KUKA KRL program: EPS_2_251349_MH86A_A_20250929014656.src

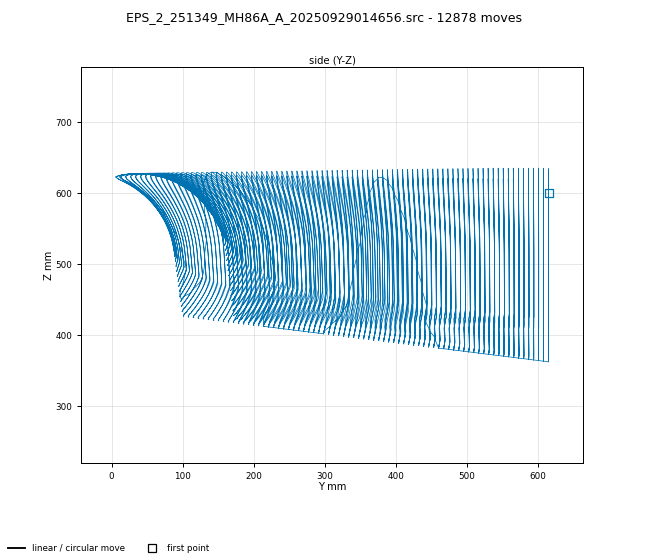
[picture p0: tool path of EPS_2_251349_MH86A_A_20250929014656.src, 12878 of 12880 moves have a stored position in this frame; points joined in program order, loops and branches not executed]
&ACCESS RVP
&REL 4
&COMMENT QRS 19112012
&PARAM EDITMASK = *
DEF PART()
EXT BAS (BAS_COMMAND :IN,REAL :IN )
INT I
BAS (#INITMOV,0 )

;KUKA QRS Post kuka4.cps  Date:22-06-2017 !

File_ID=2862

QRS_PRE_INIT()

;Init var - Until changes are made in qrs_pre_init
Outlet_Square_prg=0
Inlet_1_Square_prg=0
Inlet_2_Square_prg=0
Inlet_3_Square_prg=0
Inlet_4_Square_prg=0
Inlet_5_Square_prg=0

Outlet_1={X 0.000, Y 530.070, Z 534.500, B 0.000, E1 0.000 }
Inlet_1={X 0.000, Y 531.140, Z 519.500, B 0.000, E1 193.000 }
Outlet_1_type=201
Inlet_1_type=201
;QRS#1=Sidecore dimensions
;QRS#2=200-8" PVC SDR 35
;QRS#3=200-8" PVC SDR 35
;QRS#4=
;QRS#5=
;QRS#6=
;QRS#7=
;QRS#8=
;QRS#9=12-08 PSX
;QRS#10=12-08 PSX
;QRS#11=
;QRS#12=
;QRS#13=
;QRS#14=
;QRS#15=
;QRS#16=1220x127x914 3'
;QRS#17=EPS Height
;QRS#18=635
;QRS#19=*
;QRS#20= UPDATED VERSION 22-06-2017
;QRS#21=*
Outlet_Square=0100
Inlet_1_Square=0100
Inlet_2_Square=0
Inlet_3_Square=0
Inlet_4_Square=0
Inlet_5_Square=0
Mill_Square=1
Outlet_Square_Prg=204
Inlet_1_Square_prg=204

QRS_INIT()

$ADVANCE=5

; T1
PTP {E1 173.597,E2 173.597}
PTP {X 0,Y 615.506,A -85,B 0,C 180,E1 173.597,E2 173.597,E3 0,E4 0,E5 0,E6 0}
QRS_SPEED_INIT()
LIN {X 0,Y 615.506,Z 600,A -85,B 0,C 180,E1 173.597,E2 173.597,E3 0,E4 0,E5 0,E6 0} C_VEL
LIN {X 0,Y 615.506,Z 372.373,A -85,B 0,C 180,E1 173.597,E2 173.597} C_VEL
LIN {X 0,Y 615.506,Z 364.191,A -85,B 0,C 180,E1 173.597,E2 173.597} C_VEL
LIN {X 0,Y 615.49,Z 362.191,A -85,B 0,C 180,E1 173.411,E2 173.411} C_VEL
LIN {X 0,Y 615.479,Z 362.185,A -85,B 0,C 180,E1 170.801,E2 170.801} C_VEL
LIN {X 0,Y 615.477,Z 362.195,A -85,B 0,C 180,E1 168.139,E2 168.139} C_VEL
LIN {X 0,Y 615.49,Z 362.189,A -85,B 0,C 180,E1 165.451,E2 165.451} C_VEL
LIN {X 0,Y 615.49,Z 362.183,A -85,B 0,C 180,E1 162.73,E2 162.73} C_VEL
LIN {X 0,Y 615.493,Z 362.201,A -85,B 0,C 180,E1 159.967,E2 159.967} C_VEL
LIN {X 0,Y 615.477,Z 362.185,A -85,B 0,C 180,E1 157.155,E2 157.155} C_VEL
LIN {X 0,Y 615.493,Z 362.19,A -85,B 0,C 180,E1 154.428,E2 154.428} C_VEL
LIN {X 0,Y 615.491,Z 362.185,A -85,B 0,C 180,E1 151.547,E2 151.547} C_VEL
LIN {X 0,Y 615.483,Z 362.185,A -85,B 0,C 180,E1 148.913,E2 148.913} C_VEL
LIN {X 0,Y 615.495,Z 362.193,A -85,B 0,C 180,E1 146.463,E2 146.463} C_VEL
LIN {X 0,Y 615.488,Z 362.184,A -85,B 0,C 180,E1 143.575,E2 143.575} C_VEL
LIN {X 0,Y 615.48,Z 362.187,A -85,B 0,C 180,E1 140.938,E2 140.938} C_VEL
LIN {X 0,Y 615.494,Z 362.195,A -85,B 0,C 180,E1 138.527,E2 138.527} C_VEL
LIN {X 0,Y 615.495,Z 362.185,A -85,B 0,C 180,E1 135.851,E2 135.851} C_VEL
LIN {X 0,Y 615.481,Z 362.188,A -85,B 0,C 180,E1 133.047,E2 133.047} C_VEL
LIN {X 0,Y 615.494,Z 362.198,A -85,B 0,C 180,E1 130.605,E2 130.605} C_VEL
LIN {X 0,Y 615.489,Z 362.187,A -85,B 0,C 180,E1 128.012,E2 128.012} C_VEL
LIN {X 0,Y 615.486,Z 362.183,A -85,B 0,C 180,E1 125.615,E2 125.615} C_VEL
LIN {X 0,Y 615.478,Z 362.188,A -85,B 0,C 180,E1 123.236,E2 123.236} C_VEL
LIN {X 0,Y 615.492,Z 362.193,A -85,B 0,C 180,E1 120.919,E2 120.919} C_VEL
LIN {X 0,Y 615.483,Z 362.194,A -85,B 0,C 180,E1 118.449,E2 118.449} C_VEL
LIN {X 0,Y 615.481,Z 362.185,A -85,B 0,C 180,E1 115.567,E2 115.567} C_VEL
LIN {X 0,Y 615.489,Z 362.202,A -85,B 0,C 180,E1 112.844,E2 112.844} C_VEL
LIN {X 0,Y 615.485,Z 362.184,A -85,B 0,C 180,E1 110.033,E2 110.033} C_VEL
LIN {X 0,Y 615.479,Z 362.193,A -85,B 0,C 180,E1 107.271,E2 107.271} C_VEL
LIN {X 0,Y 615.479,Z 362.191,A -85,B 0,C 180,E1 104.549,E2 104.549} C_VEL
LIN {X 0,Y 615.489,Z 362.183,A -85,B 0,C 180,E1 101.861,E2 101.861} C_VEL
LIN {X 0,Y 615.49,Z 362.198,A -85,B 0,C 180,E1 99.199,E2 99.199} C_VEL
LIN {X 0,Y 615.499,Z 362.314,A -85,B 0,C 180,E1 97.058,E2 97.058} C_VEL
LIN {X 0,Y 615.484,Z 376.753,A -85,B 0,C 180,E1 94.749,E2 94.749} C_VEL
LIN {X 0,Y 615.497,Z 394.683,A -85,B 0,C 180,E1 91.963,E2 91.963} C_VEL
LIN {X 0,Y 615.488,Z 408.592,A -85,B 0,C 180,E1 89.857,E2 89.857} C_VEL
LIN {X 0,Y 615.485,Z 410.307,A -85,B 0,C 180,E1 89.796,E2 89.796} C_VEL
LIN {X 0,Y 615.497,Z 515.58,A -85,B 0,C 180,E1 88.548,E2 88.548} C_VEL
LIN {X 0,Y 615.498,Z 527.992,A -85,B 0,C 180,E1 88.283,E2 88.283} C_VEL
LIN {X 0,Y 615.498,Z 540.764,A -85,B 0,C 180,E1 87.873,E2 87.873} C_VEL
LIN {X 0,Y 615.486,Z 552.111,A -85,B 0,C 180,E1 87.382,E2 87.382} C_VEL
LIN {X 0,Y 615.484,Z 563.831,A -85,B 0,C 180,E1 86.727,E2 86.727} C_VEL
LIN {X 0,Y 615.498,Z 574.262,A -85,B 0,C 180,E1 85.99,E2 85.99} C_VEL
LIN {X 0,Y 615.497,Z 584.574,A -85,B 0,C 180,E1 85.088,E2 85.088} C_VEL
LIN {X 0,Y 615.499,Z 593.527,A -85,B 0,C 180,E1 84.102,E2 84.102} C_VEL
LIN {X 0,Y 615.497,Z 600.873,A -85,B 0,C 180,E1 83.1,E2 83.1} C_VEL
LIN {X 0,Y 615.497,Z 606.596,A -85,B 0,C 180,E1 82.125,E2 82.125} C_VEL
LIN {X 0,Y 615.497,Z 611.188,A -85,B 0,C 180,E1 81.133,E2 81.133} C_VEL
LIN {X 0,Y 615.498,Z 614.685,A -85,B 0,C 180,E1 80.138,E2 80.138} C_VEL
LIN {X 0,Y 615.494,Z 617.25,A -85,B 0,C 180,E1 79.109,E2 79.109} C_VEL
LIN {X 0,Y 615.496,Z 618.726,A -85,B 0,C 180,E1 78.14,E2 78.14} C_VEL
LIN {X 0,Y 615.497,Z 619.266,A -85,B 0,C 180,E1 77.47,E2 77.47} C_VEL
LIN {X 0,Y 615.496,Z 619.357,A -85,B 0,C 180,E1 76.799,E2 76.799} C_VEL
LIN {X 0,Y 615.496,Z 619.007,A -85,B 0,C 180,E1 76.065,E2 76.065} C_VEL
LIN {X 0,Y 615.495,Z 618.351,A -85,B 0,C 180,E1 75.452,E2 75.452} C_VEL
LIN {X 0,Y 615.495,Z 617.194,A -85,B 0,C 180,E1 74.775,E2 74.775} C_VEL
LIN {X 0,Y 615.493,Z 614.033,A -85,B 0,C 180,E1 73.568,E2 73.568} C_VEL
LIN {X 0,Y 615.499,Z 609.514,A -85,B 0,C 180,E1 72.387,E2 72.387} C_VEL
LIN {X 0,Y 615.496,Z 604.234,A -85,B 0,C 180,E1 71.355,E2 71.355} C_VEL
LIN {X 0,Y 615.496,Z 597.453,A -85,B 0,C 180,E1 70.316,E2 70.316} C_VEL
LIN {X 0,Y 615.494,Z 588.884,A -85,B 0,C 180,E1 69.27,E2 69.27} C_VEL
LIN {X 0,Y 615.497,Z 579.965,A -85,B 0,C 180,E1 68.393,E2 68.393} C_VEL
LIN {X 0,Y 615.495,Z 568.994,A -85,B 0,C 180,E1 67.528,E2 67.528} C_VEL
LIN {X 0,Y 615.484,Z 558.946,A -85,B 0,C 180,E1 66.89,E2 66.89} C_VEL
LIN {X 0,Y 615.5,Z 546.63,A -85,B 0,C 180,E1 66.274,E2 66.274} C_VEL
LIN {X 0,Y 615.497,Z 533.761,A -85,B 0,C 180,E1 65.794,E2 65.794} C_VEL
LIN {X 0,Y 615.495,Z 520.923,A -85,B 0,C 180,E1 65.46,E2 65.46} C_VEL
LIN {X 0,Y 615.497,Z 505.869,A -85,B 0,C 180,E1 65.235,E2 65.235} C_VEL
LIN {X 0,Y 615.487,Z 409.668,A -85,B 0,C 180,E1 64.103,E2 64.103} C_VEL
LIN {X 0,Y 615.488,Z 408.193,A -85,B 0,C 180,E1 64.012,E2 64.012} C_VEL
LIN {X 0,Y 615.498,Z 389.57,A -85,B 0,C 180,E1 61.157,E2 61.157} C_VEL
LIN {X 0,Y 615.488,Z 371.358,A -85,B 0,C 180,E1 58.316,E2 58.316} C_VEL
LIN {X 0,Y 615.493,Z 362.338,A -85,B 0,C 180,E1 56.863,E2 56.863} C_VEL
LIN {X 0,Y 615.489,Z 362.184,A -85,B 0,C 180,E1 54.166,E2 54.166} C_VEL
LIN {X 0,Y 615.482,Z 362.184,A -85,B 0,C 180,E1 51.932,E2 51.932} C_VEL
LIN {X 0,Y 615.483,Z 362.187,A -85,B 0,C 180,E1 49.394,E2 49.394} C_VEL
LIN {X 0,Y 615.495,Z 362.197,A -85,B 0,C 180,E1 46.757,E2 46.757} C_VEL
LIN {X 0,Y 615.482,Z 362.184,A -85,B 0,C 180,E1 43.998,E2 43.998} C_VEL
LIN {X 0,Y 615.485,Z 362.186,A -85,B 0,C 180,E1 41.474,E2 41.474} C_VEL
LIN {X 0,Y 615.497,Z 362.2,A -85,B 0,C 180,E1 38.904,E2 38.904} C_VEL
LIN {X 0,Y 615.493,Z 362.186,A -85,B 0,C 180,E1 36.424,E2 36.424} C_VEL
LIN {X 0,Y 615.484,Z 362.186,A -85,B 0,C 180,E1 33.536,E2 33.536} C_VEL
LIN {X 0,Y 615.493,Z 362.2,A -85,B 0,C 180,E1 30.919,E2 30.919} C_VEL
LIN {X 0,Y 615.495,Z 362.185,A -85,B 0,C 180,E1 28.454,E2 28.454} C_VEL
LIN {X 0,Y 615.479,Z 362.186,A -85,B 0,C 180,E1 25.716,E2 25.716} C_VEL
LIN {X 0,Y 615.489,Z 362.196,A -85,B 0,C 180,E1 22.844,E2 22.844} C_VEL
LIN {X 0,Y 615.479,Z 362.184,A -85,B 0,C 180,E1 20.033,E2 20.033} C_VEL
LIN {X 0,Y 615.496,Z 362.193,A -85,B 0,C 180,E1 17.27,E2 17.27} C_VEL
LIN {X 0,Y 615.493,Z 362.186,A -85,B 0,C 180,E1 14.549,E2 14.549} C_VEL
LIN {X 0,Y 615.476,Z 362.186,A -85,B 0,C 180,E1 11.861,E2 11.861} C_VEL
LIN {X 0,Y 615.496,Z 362.198,A -85,B 0,C 180,E1 9.199,E2 9.199} C_VEL
LIN {X 0,Y 615.495,Z 362.184,A -85,B 0,C 180,E1 6.557,E2 6.557} C_VEL
LIN {X 0,Y 615.476,Z 362.186,A -85,B 0,C 180,E1 3.929,E2 3.929} C_VEL
LIN {X 0,Y 615.496,Z 362.195,A -85,B 0,C 180,E1 1.309,E2 1.309} C_VEL
LIN {X 0,Y 615.491,Z 362.187,A -85,B 0,C 180,E1 -1.309,E2 -1.309} C_VEL
LIN {X 0,Y 615.476,Z 362.185,A -85,B 0,C 180,E1 -3.929,E2 -3.929} C_VEL
LIN {X 0,Y 615.497,Z 362.194,A -85,B 0,C 180,E1 -6.598,E2 -6.598} C_VEL
LIN {X 0,Y 615.486,Z 362.189,A -85,B 0,C 180,E1 -9.199,E2 -9.199} C_VEL
LIN {X 0,Y 615.478,Z 362.185,A -85,B 0,C 180,E1 -11.861,E2 -11.861} C_VEL
LIN {X 0,Y 615.497,Z 362.194,A -85,B 0,C 180,E1 -14.549,E2 -14.549} C_VEL
LIN {X 0,Y 615.493,Z 362.185,A -85,B 0,C 180,E1 -17.27,E2 -17.27} C_VEL
LIN {X 0,Y 615.479,Z 362.186,A -85,B 0,C 180,E1 -20.033,E2 -20.033} C_VEL
LIN {X 0,Y 615.492,Z 362.196,A -85,B 0,C 180,E1 -22.844,E2 -22.844} C_VEL
LIN {X 0,Y 615.477,Z 362.184,A -85,B 0,C 180,E1 -25.716,E2 -25.716} C_VEL
LIN {X 0,Y 615.497,Z 362.194,A -85,B 0,C 180,E1 -28.454,E2 -28.454} C_VEL
LIN {X 0,Y 615.49,Z 362.188,A -85,B 0,C 180,E1 -31.089,E2 -31.089} C_VEL
LIN {X 0,Y 615.484,Z 362.183,A -85,B 0,C 180,E1 -33.536,E2 -33.536} C_VEL
LIN {X 0,Y 615.495,Z 362.195,A -85,B 0,C 180,E1 -36.424,E2 -36.424} C_VEL
LIN {X 0,Y 615.488,Z 362.188,A -85,B 0,C 180,E1 -39.064,E2 -39.064} C_VEL
LIN {X 0,Y 615.485,Z 362.183,A -85,B 0,C 180,E1 -41.474,E2 -41.474} C_VEL
LIN {X 0,Y 615.491,Z 362.189,A -85,B 0,C 180,E1 -44.149,E2 -44.149} C_VEL
LIN {X 0,Y 615.489,Z 362.189,A -85,B 0,C 180,E1 -46.953,E2 -46.953} C_VEL
LIN {X 0,Y 615.482,Z 362.183,A -85,B 0,C 180,E1 -49.394,E2 -49.394} C_VEL
LIN {X 0,Y 615.484,Z 362.188,A -85,B 0,C 180,E1 -51.989,E2 -51.989} C_VEL
LIN {X 0,Y 615.496,Z 362.198,A -85,B 0,C 180,E1 -54.386,E2 -54.386} C_VEL
LIN {X 0,Y 615.488,Z 362.192,A -85,B 0,C 180,E1 -56.765,E2 -56.765} C_VEL
LIN {X 0,Y 615.495,Z 362.183,A -85,B 0,C 180,E1 -59.082,E2 -59.082} C_VEL
LIN {X 0,Y 615.477,Z 362.185,A -85,B 0,C 180,E1 -61.552,E2 -61.552} C_VEL
LIN {X 0,Y 615.498,Z 362.2,A -85,B 0,C 180,E1 -64.43,E2 -64.43} C_VEL
LIN {X 0,Y 615.488,Z 362.183,A -85,B 0,C 180,E1 -67.156,E2 -67.156} C_VEL
LIN {X 0,Y 615.495,Z 362.441,A -85,B 0,C 180,E1 -68.481,E2 -68.481} C_VEL
LIN {X 0,Y 615.495,Z 380.964,A -85,B 0,C 180,E1 -71.182,E2 -71.182} C_VEL
LIN {X 0,Y 615.489,Z 401.427,A -85,B 0,C 180,E1 -74.095,E2 -74.095} C_VEL
LIN {X 0,Y 615.497,Z 422.521,A -85,B 0,C 180,E1 -77.051,E2 -77.051} C_VEL
LIN {X 0,Y 615.497,Z 423.747,A -85,B 0,C 180,E1 -77.135,E2 -77.135} C_VEL
LIN {X 0,Y 615.498,Z 530.85,A -85,B 0,C 180,E1 -78.411,E2 -78.411} C_VEL
LIN {X 0,Y 615.498,Z 543.356,A -85,B 0,C 180,E1 -78.682,E2 -78.682} C_VEL
LIN {X 0,Y 615.496,Z 556.503,A -85,B 0,C 180,E1 -79.109,E2 -79.109} C_VEL
LIN {X 0,Y 615.483,Z 568.485,A -85,B 0,C 180,E1 -79.64,E2 -79.64} C_VEL
LIN {X 0,Y 615.487,Z 580.001,A -85,B 0,C 180,E1 -80.304,E2 -80.304} C_VEL
LIN {X 0,Y 615.499,Z 590.345,A -85,B 0,C 180,E1 -81.05,E2 -81.05} C_VEL
LIN {X 0,Y 615.497,Z 598.815,A -85,B 0,C 180,E1 -81.794,E2 -81.794} C_VEL
LIN {X 0,Y 615.498,Z 606.609,A -85,B 0,C 180,E1 -82.62,E2 -82.62} C_VEL
LIN {X 0,Y 615.496,Z 614.205,A -85,B 0,C 180,E1 -83.608,E2 -83.608} C_VEL
LIN {X 0,Y 615.499,Z 621.206,A -85,B 0,C 180,E1 -84.759,E2 -84.759} C_VEL
LIN {X 0,Y 615.493,Z 625.853,A -85,B 0,C 180,E1 -85.744,E2 -85.744} C_VEL
LIN {X 0,Y 615.495,Z 629.399,A -85,B 0,C 180,E1 -86.727,E2 -86.727} C_VEL
LIN {X 0,Y 615.497,Z 631.233,A -85,B 0,C 180,E1 -87.382,E2 -87.382} C_VEL
LIN {X 0,Y 615.497,Z 632.608,A -85,B 0,C 180,E1 -88.037,E2 -88.037} C_VEL
LIN {X 0,Y 615.496,Z 634.174,A -85,B 0,C 180,E1 -89.346,E2 -89.346} C_VEL
LIN {X 0,Y 615.494,Z 634.389,A -85,B 0,C 180,E1 -90,E2 -90} C_VEL
LIN {X 0,Y 615.496,Z 633.58,A -85,B 0,C 180,E1 -91.309,E2 -91.309} C_VEL
LIN {X 0,Y 615.497,Z 632.608,A -85,B 0,C 180,E1 -91.963,E2 -91.963} C_VEL
LIN {X 0,Y 615.497,Z 631.233,A -85,B 0,C 180,E1 -92.618,E2 -92.618} C_VEL
LIN {X 0,Y 615.496,Z 628.349,A -85,B 0,C 180,E1 -93.601,E2 -93.601} C_VEL
LIN {X 0,Y 615.498,Z 624.441,A -85,B 0,C 180,E1 -94.585,E2 -94.585} C_VEL
LIN {X 0,Y 615.499,Z 619.405,A -85,B 0,C 180,E1 -95.57,E2 -95.57} C_VEL
LIN {X 0,Y 615.497,Z 612.87,A -85,B 0,C 180,E1 -96.583,E2 -96.583} C_VEL
LIN {X 0,Y 615.497,Z 605.133,A -85,B 0,C 180,E1 -97.545,E2 -97.545} C_VEL
LIN {X 0,Y 615.498,Z 597.045,A -85,B 0,C 180,E1 -98.371,E2 -98.371} C_VEL
LIN {X 0,Y 615.499,Z 587.168,A -85,B 0,C 180,E1 -99.199,E2 -99.199} C_VEL
LIN {X 0,Y 615.487,Z 575.982,A -85,B 0,C 180,E1 -99.945,E2 -99.945} C_VEL
LIN {X 0,Y 615.486,Z 565.024,A -85,B 0,C 180,E1 -100.527,E2 -100.527} C_VEL
LIN {X 0,Y 615.499,Z 552.418,A -85,B 0,C 180,E1 -101.042,E2 -101.042} C_VEL
LIN {X 0,Y 615.499,Z 540.066,A -85,B 0,C 180,E1 -101.401,E2 -101.401} C_VEL
LIN {X 0,Y 615.499,Z 526.468,A -85,B 0,C 180,E1 -101.652,E2 -101.652} C_VEL
LIN {X 0,Y 615.496,Z 423.736,A -85,B 0,C 180,E1 -102.865,E2 -102.865} C_VEL
LIN {X 0,Y 615.497,Z 422.518,A -85,B 0,C 180,E1 -102.949,E2 -102.949} C_VEL
LIN {X 0,Y 615.489,Z 401.425,A -85,B 0,C 180,E1 -105.905,E2 -105.905} C_VEL
LIN {X 0,Y 615.495,Z 380.962,A -85,B 0,C 180,E1 -108.818,E2 -108.818} C_VEL
LIN {X 0,Y 615.496,Z 362.439,A -85,B 0,C 180,E1 -111.519,E2 -111.519} C_VEL
LIN {X 0,Y 615.488,Z 362.184,A -85,B 0,C 180,E1 -112.844,E2 -112.844} C_VEL
LIN {X 0,Y 615.498,Z 362.194,A -85,B 0,C 180,E1 -115.715,E2 -115.715} C_VEL
LIN {X 0,Y 615.477,Z 362.185,A -85,B 0,C 180,E1 -118.448,E2 -118.448} C_VEL
LIN {X 0,Y 615.492,Z 362.19,A -85,B 0,C 180,E1 -121.086,E2 -121.086} C_VEL
LIN {X 0,Y 615.484,Z 362.186,A -85,B 0,C 180,E1 -124.022,E2 -124.022} C_VEL
LIN {X 0,Y 615.479,Z 362.185,A -85,B 0,C 180,E1 -126.425,E2 -126.425} C_VEL
LIN {X 0,Y 615.493,Z 362.193,A -85,B 0,C 180,E1 -129.062,E2 -129.062} C_VEL
LIN {X 0,Y 615.494,Z 362.194,A -85,B 0,C 180,E1 -131.472,E2 -131.472} C_VEL
LIN {X 0,Y 615.478,Z 362.185,A -85,B 0,C 180,E1 -134.149,E2 -134.149} C_VEL
LIN {X 0,Y 615.494,Z 362.194,A -85,B 0,C 180,E1 -136.951,E2 -136.951} C_VEL
LIN {X 0,Y 615.486,Z 362.184,A -85,B 0,C 180,E1 -139.91,E2 -139.91} C_VEL
LIN {X 0,Y 615.494,Z 362.191,A -85,B 0,C 180,E1 -142.758,E2 -142.758} C_VEL
LIN {X 0,Y 615.49,Z 362.192,A -85,B 0,C 180,E1 -145.298,E2 -145.298} C_VEL
LIN {X 0,Y 615.493,Z 362.183,A -85,B 0,C 180,E1 -147.667,E2 -147.667} C_VEL
LIN {X 0,Y 615.489,Z 362.192,A -85,B 0,C 180,E1 -150.594,E2 -150.594} C_VEL
LIN {X 0,Y 615.493,Z 362.183,A -85,B 0,C 180,E1 -153.556,E2 -153.556} C_VEL
LIN {X 0,Y 615.485,Z 362.191,A -85,B 0,C 180,E1 -156.443,E2 -156.443} C_VEL
LIN {X 0,Y 615.479,Z 362.189,A -85,B 0,C 180,E1 -159.269,E2 -159.269} C_VEL
LIN {X 0,Y 615.477,Z 362.187,A -85,B 0,C 180,E1 -162.043,E2 -162.043} C_VEL
LIN {X 0,Y 615.486,Z 362.199,A -85,B 0,C 180,E1 -164.774,E2 -164.774} C_VEL
LIN {X 0,Y 615.484,Z 362.184,A -85,B 0,C 180,E1 -167.47,E2 -167.47} C_VEL
LIN {X 0,Y 615.477,Z 362.192,A -85,B 0,C 180,E1 -170.138,E2 -170.138} C_VEL
LIN {X 0,Y 615.483,Z 362.194,A -85,B 0,C 180,E1 -172.784,E2 -172.784} C_VEL
LIN {X 0,Y 615.491,Z 362.182,A -85,B 0,C 180,E1 -175.415,E2 -175.415} C_VEL
LIN {X 0,Y 615.478,Z 362.193,A -85,B 0,C 180,E1 -178.037,E2 -178.037} C_VEL
LIN {X 0,Y 615.484,Z 362.194,A -85,B 0,C 180,E1 -180.654,E2 -180.654} C_VEL
LIN {X 0,Y 615.485,Z 362.183,A -85,B 0,C 180,E1 -183.273,E2 -183.273} C_VEL
LIN {X 0,Y 615.481,Z 362.192,A -85,B 0,C 180,E1 -185.899,E2 -185.899} C_VEL
LIN {X 0,Y 615.49,Z 362.191,A -85,B 0,C 180,E1 -186.589,E2 -186.589} C_VEL
LIN {X 0,Y 614.809,Z 362.332,A -85,B 0,C 180,E1 -187.135,E2 -187.135} C_VEL
LIN {X 0,Y 611.969,Z 362.756,A -85,B 0,C 180,E1 -188.021,E2 -188.021} C_VEL
LIN {X 0,Y 609.575,Z 363.062,A -85,B 0,C 180,E1 -188.733,E2 -188.733} C_VEL
LIN {X 0,Y 608.54,Z 363.178,A -85,B 0,C 180,E1 -189.283,E2 -189.283} C_VEL
LIN {X 0,Y 608.452,Z 363.188,A -85,B 0,C 180,E1 -189.469,E2 -189.469} C_VEL
LIN {X 0,Y 608.455,Z 363.195,A -85,B 0,C 180,E1 -192,E2 -192} C_VEL
LIN {X 0,Y 608.476,Z 363.186,A -85,B 0,C 180,E1 -194.72,E2 -194.72} C_VEL
LIN {X 0,Y 608.456,Z 363.189,A -85,B 0,C 180,E1 -197.476,E2 -197.476} C_VEL
LIN {X 0,Y 608.466,Z 363.192,A -85,B 0,C 180,E1 -200.274,E2 -200.274} C_VEL
LIN {X 0,Y 608.457,Z 363.19,A -85,B 0,C 180,E1 -202.478,E2 -202.478} C_VEL
LIN {X 0,Y 608.453,Z 363.189,A -85,B 0,C 180,E1 -204.571,E2 -204.571} C_VEL
LIN {X 0,Y 608.474,Z 363.186,A -85,B 0,C 180,E1 -207.208,E2 -207.208} C_VEL
LIN {X 0,Y 608.475,Z 363.193,A -85,B 0,C 180,E1 -209.974,E2 -209.974} C_VEL
LIN {X 0,Y 608.463,Z 363.187,A -85,B 0,C 180,E1 -212.524,E2 -212.524} C_VEL
LIN {X 0,Y 608.443,Z 363.192,A -85,B 0,C 180,E1 -215.278,E2 -215.278} C_VEL
LIN {X 0,Y 608.473,Z 363.195,A -85,B 0,C 180,E1 -217.746,E2 -217.746} C_VEL
LIN {X 0,Y 608.451,Z 363.189,A -85,B 0,C 180,E1 -220.33,E2 -220.33} C_VEL
LIN {X 0,Y 608.453,Z 363.189,A -85,B 0,C 180,E1 -222.96,E2 -222.96} C_VEL
LIN {X 0,Y 608.458,Z 363.194,A -85,B 0,C 180,E1 -225.736,E2 -225.736} C_VEL
LIN {X 0,Y 608.457,Z 363.187,A -85,B 0,C 180,E1 -228.658,E2 -228.658} C_VEL
LIN {X 0,Y 608.47,Z 363.195,A -85,B 0,C 180,E1 -231.413,E2 -231.413} C_VEL
LIN {X 0,Y 608.478,Z 363.187,A -85,B 0,C 180,E1 -233.951,E2 -233.951} C_VEL
LIN {X 0,Y 608.464,Z 363.186,A -85,B 0,C 180,E1 -236.33,E2 -236.33} C_VEL
LIN {X 0,Y 608.46,Z 363.188,A -85,B 0,C 180,E1 -238.731,E2 -238.731} C_VEL
LIN {X 0,Y 608.475,Z 363.194,A -85,B 0,C 180,E1 -241.38,E2 -241.38} C_VEL
LIN {X 0,Y 608.471,Z 363.185,A -85,B 0,C 180,E1 -244.279,E2 -244.279} C_VEL
LIN {X 0,Y 608.45,Z 363.193,A -85,B 0,C 180,E1 -246.876,E2 -246.876} C_VEL
LIN {X 0,Y 608.46,Z 363.188,A -85,B 0,C 180,E1 -249.726,E2 -249.726} C_VEL
LIN {X 0,Y 608.451,Z 363.19,A -85,B 0,C 180,E1 -252.524,E2 -252.524} C_VEL
LIN {X 0,Y 608.47,Z 363.191,A -85,B 0,C 180,E1 -255.28,E2 -255.28} C_VEL
LIN {X 0,Y 608.462,Z 363.186,A -85,B 0,C 180,E1 -258,E2 -258} C_VEL
LIN {X 0,Y 608.474,Z 363.191,A -85,B 0,C 180,E1 -260.694,E2 -260.694} C_VEL
LIN {X 0,Y 608.486,Z 363.376,A -85,B 0,C 180,E1 -262.889,E2 -262.889} C_VEL
LIN {X 0,Y 608.498,Z 377.808,A -85,B 0,C 180,E1 -265.197,E2 -265.197} C_VEL
LIN {X 0,Y 608.499,Z 395.794,A -85,B 0,C 180,E1 -268.014,E2 -268.014} C_VEL
LIN {X 0,Y 608.48,Z 408.761,A -85,B 0,C 180,E1 -270,E2 -270} C_VEL
LIN {X 0,Y 608.563,Z 410.777,A -85,B 0,C 180,E1 -270.062,E2 -270.062} C_VEL
LIN {X 0,Y 608.557,Z 516.027,A -85,B 0,C 180,E1 -271.323,E2 -271.323} C_VEL
LIN {X 0,Y 608.56,Z 529.053,A -85,B 0,C 180,E1 -271.613,E2 -271.613} C_VEL
LIN {X 0,Y 608.519,Z 541.614,A -85,B 0,C 180,E1 -272.027,E2 -272.027} C_VEL
LIN {X 0,Y 608.512,Z 553.646,A -85,B 0,C 180,E1 -272.565,E2 -272.565} C_VEL
LIN {X 0,Y 608.483,Z 565.068,A -85,B 0,C 180,E1 -273.228,E2 -273.228} C_VEL
LIN {X 0,Y 608.472,Z 575.378,A -85,B 0,C 180,E1 -273.974,E2 -273.974} C_VEL
LIN {X 0,Y 608.464,Z 584.735,A -85,B 0,C 180,E1 -274.803,E2 -274.803} C_VEL
LIN {X 0,Y 608.459,Z 593.778,A -85,B 0,C 180,E1 -275.8,E2 -275.8} C_VEL
LIN {X 0,Y 608.461,Z 601.1,A -85,B 0,C 180,E1 -276.799,E2 -276.799} C_VEL
LIN {X 0,Y 608.45,Z 606.08,A -85,B 0,C 180,E1 -277.633,E2 -277.633} C_VEL
LIN {X 0,Y 608.427,Z 610.93,A -85,B 0,C 180,E1 -278.636,E2 -278.636} C_VEL
LIN {X 0,Y 608.429,Z 614.661,A -85,B 0,C 180,E1 -279.642,E2 -279.642} C_VEL
LIN {X 0,Y 608.45,Z 618.005,A -85,B 0,C 180,E1 -280.946,E2 -280.946} C_VEL
LIN {X 0,Y 608.44,Z 619.506,A -85,B 0,C 180,E1 -282,E2 -282} C_VEL
LIN {X 0,Y 608.418,Z 619.92,A -85,B 0,C 180,E1 -282.678,E2 -282.678} C_VEL
LIN {X 0,Y 608.442,Z 619.573,A -85,B 0,C 180,E1 -284.006,E2 -284.006} C_VEL
LIN {X 0,Y 608.418,Z 618.715,A -85,B 0,C 180,E1 -284.721,E2 -284.721} C_VEL
LIN {X 0,Y 608.419,Z 617.443,A -85,B 0,C 180,E1 -285.407,E2 -285.407} C_VEL
LIN {X 0,Y 608.424,Z 614.45,A -85,B 0,C 180,E1 -286.515,E2 -286.515} C_VEL
LIN {X 0,Y 608.429,Z 610.832,A -85,B 0,C 180,E1 -287.477,E2 -287.477} C_VEL
LIN {X 0,Y 608.443,Z 606.182,A -85,B 0,C 180,E1 -288.438,E2 -288.438} C_VEL
LIN {X 0,Y 608.451,Z 599.223,A -85,B 0,C 180,E1 -289.57,E2 -289.57} C_VEL
LIN {X 0,Y 608.459,Z 591.706,A -85,B 0,C 180,E1 -290.54,E2 -290.54} C_VEL
LIN {X 0,Y 608.467,Z 582.342,A -85,B 0,C 180,E1 -291.513,E2 -291.513} C_VEL
LIN {X 0,Y 608.491,Z 572.867,A -85,B 0,C 180,E1 -292.315,E2 -292.315} C_VEL
LIN {X 0,Y 608.493,Z 562.413,A -85,B 0,C 180,E1 -293.032,E2 -293.032} C_VEL
LIN {X 0,Y 608.501,Z 550.841,A -85,B 0,C 180,E1 -293.662,E2 -293.662} C_VEL
LIN {X 0,Y 608.536,Z 538.912,A -85,B 0,C 180,E1 -294.164,E2 -294.164} C_VEL
LIN {X 0,Y 608.553,Z 526.432,A -85,B 0,C 180,E1 -294.549,E2 -294.549} C_VEL
LIN {X 0,Y 608.551,Z 514.31,A -85,B 0,C 180,E1 -294.794,E2 -294.794} C_VEL
LIN {X 0,Y 608.532,Z 409.381,A -85,B 0,C 180,E1 -296.054,E2 -296.054} C_VEL
LIN {X 0,Y 608.468,Z 408.44,A -85,B 0,C 180,E1 -296.126,E2 -296.126} C_VEL
LIN {X 0,Y 608.494,Z 391.257,A -85,B 0,C 180,E1 -298.783,E2 -298.783} C_VEL
LIN {X 0,Y 608.514,Z 373.926,A -85,B 0,C 180,E1 -301.507,E2 -301.507} C_VEL
LIN {X 0,Y 608.471,Z 363.297,A -85,B 0,C 180,E1 -303.223,E2 -303.223} C_VEL
LIN {X 0,Y 608.475,Z 363.185,A -85,B 0,C 180,E1 -306.049,E2 -306.049} C_VEL
LIN {X 0,Y 608.472,Z 363.187,A -85,B 0,C 180,E1 -308.587,E2 -308.587} C_VEL
LIN {X 0,Y 608.467,Z 363.193,A -85,B 0,C 180,E1 -311.343,E2 -311.343} C_VEL
LIN {X 0,Y 608.449,Z 363.188,A -85,B 0,C 180,E1 -314.263,E2 -314.263} C_VEL
LIN {X 0,Y 608.463,Z 363.196,A -85,B 0,C 180,E1 -317.041,E2 -317.041} C_VEL
LIN {X 0,Y 608.454,Z 363.189,A -85,B 0,C 180,E1 -319.697,E2 -319.697} C_VEL
LIN {X 0,Y 608.468,Z 363.185,A -85,B 0,C 180,E1 -322.254,E2 -322.254} C_VEL
LIN {X 0,Y 608.482,Z 363.194,A -85,B 0,C 180,E1 -325.088,E2 -325.088} C_VEL
LIN {X 0,Y 608.467,Z 363.186,A -85,B 0,C 180,E1 -327.906,E2 -327.906} C_VEL
LIN {X 0,Y 608.462,Z 363.186,A -85,B 0,C 180,E1 -330.22,E2 -330.22} C_VEL
LIN {X 0,Y 608.485,Z 363.19,A -85,B 0,C 180,E1 -332.789,E2 -332.789} C_VEL
LIN {X 0,Y 608.456,Z 363.19,A -85,B 0,C 180,E1 -335.429,E2 -335.429} C_VEL
LIN {X 0,Y 608.47,Z 363.186,A -85,B 0,C 180,E1 -338.308,E2 -338.308} C_VEL
LIN {X 0,Y 608.47,Z 363.19,A -85,B 0,C 180,E1 -341.28,E2 -341.28} C_VEL
LIN {X 0,Y 608.456,Z 363.187,A -85,B 0,C 180,E1 -343.906,E2 -343.906} C_VEL
LIN {X 0,Y 608.468,Z 363.191,A -85,B 0,C 180,E1 -346.644,E2 -346.644} C_VEL
LIN {X 0,Y 608.472,Z 363.188,A -85,B 0,C 180,E1 -349.35,E2 -349.35} C_VEL
LIN {X 0,Y 608.47,Z 363.185,A -85,B 0,C 180,E1 -352.033,E2 -352.033} C_VEL
LIN {X 0,Y 608.472,Z 363.192,A -85,B 0,C 180,E1 -354.698,E2 -354.698} C_VEL
LIN {X 0,Y 608.483,Z 363.186,A -85,B 0,C 180,E1 -357.352,E2 -357.352} C_VEL
LIN {X 0,Y 608.468,Z 363.185,A -85,B 0,C 180,E1 -360,E2 -360} C_VEL
LIN {X 0,Y 608.486,Z 363.191,A -85,B 0,C 180,E1 -362.648,E2 -362.648} C_VEL
LIN {X 0,Y 608.468,Z 363.188,A -85,B 0,C 180,E1 -365.302,E2 -365.302} C_VEL
LIN {X 0,Y 608.471,Z 363.185,A -85,B 0,C 180,E1 -367.967,E2 -367.967} C_VEL
LIN {X 0,Y 608.474,Z 363.193,A -85,B 0,C 180,E1 -370.65,E2 -370.65} C_VEL
LIN {X 0,Y 608.464,Z 363.187,A -85,B 0,C 180,E1 -373.357,E2 -373.357} C_VEL
LIN {X 0,Y 608.457,Z 363.188,A -85,B 0,C 180,E1 -376.094,E2 -376.094} C_VEL
LIN {X 0,Y 608.456,Z 363.195,A -85,B 0,C 180,E1 -378.87,E2 -378.87} C_VEL
LIN {X 0,Y 608.47,Z 363.185,A -85,B 0,C 180,E1 -381.692,E2 -381.692} C_VEL
LIN {X 0,Y 608.454,Z 363.196,A -85,B 0,C 180,E1 -384.571,E2 -384.571} C_VEL
LIN {X 0,Y 608.477,Z 363.186,A -85,B 0,C 180,E1 -387.21,E2 -387.21} C_VEL
LIN {X 0,Y 608.46,Z 363.187,A -85,B 0,C 180,E1 -389.973,E2 -389.973} C_VEL
LIN {X 0,Y 608.467,Z 363.195,A -85,B 0,C 180,E1 -392.525,E2 -392.525} C_VEL
LIN {X 0,Y 608.441,Z 363.19,A -85,B 0,C 180,E1 -395.278,E2 -395.278} C_VEL
LIN {X 0,Y 608.468,Z 363.185,A -85,B 0,C 180,E1 -397.747,E2 -397.747} C_VEL
LIN {X 0,Y 608.476,Z 363.191,A -85,B 0,C 180,E1 -400.333,E2 -400.333} C_VEL
LIN {X 0,Y 608.483,Z 363.184,A -85,B 0,C 180,E1 -403.312,E2 -403.312} C_VEL
LIN {X 0,Y 608.469,Z 363.189,A -85,B 0,C 180,E1 -406.132,E2 -406.132} C_VEL
LIN {X 0,Y 608.46,Z 363.192,A -85,B 0,C 180,E1 -408.825,E2 -408.825} C_VEL
LIN {X 0,Y 608.47,Z 363.185,A -85,B 0,C 180,E1 -411.413,E2 -411.413} C_VEL
LIN {X 0,Y 608.476,Z 363.187,A -85,B 0,C 180,E1 -413.951,E2 -413.951} C_VEL
LIN {X 0,Y 608.471,Z 363.193,A -85,B 0,C 180,E1 -416.331,E2 -416.331} C_VEL
LIN {X 0,Y 608.479,Z 363.19,A -85,B 0,C 180,E1 -418.728,E2 -418.728} C_VEL
LIN {X 0,Y 608.469,Z 363.185,A -85,B 0,C 180,E1 -421.381,E2 -421.381} C_VEL
LIN {X 0,Y 608.449,Z 363.191,A -85,B 0,C 180,E1 -423.965,E2 -423.965} C_VEL
LIN {X 0,Y 608.468,Z 363.192,A -85,B 0,C 180,E1 -426.156,E2 -426.156} C_VEL
LIN {X 0,Y 608.509,Z 363.352,A -85,B 0,C 180,E1 -428.355,E2 -428.355} C_VEL
LIN {X 0,Y 608.545,Z 378.582,A -85,B 0,C 180,E1 -430.609,E2 -430.609} C_VEL
LIN {X 0,Y 608.487,Z 396.681,A -85,B 0,C 180,E1 -433.217,E2 -433.217} C_VEL
LIN {X 0,Y 608.503,Z 416.976,A -85,B 0,C 180,E1 -436.104,E2 -436.104} C_VEL
LIN {X 0,Y 608.507,Z 423.299,A -85,B 0,C 180,E1 -436.964,E2 -436.964} C_VEL
LIN {X 0,Y 608.573,Z 428.545,A -85,B 0,C 180,E1 -437.05,E2 -437.05} C_VEL
LIN {X 0,Y 608.549,Z 530.969,A -85,B 0,C 180,E1 -438.277,E2 -438.277} C_VEL
LIN {X 0,Y 608.547,Z 544.231,A -85,B 0,C 180,E1 -438.573,E2 -438.573} C_VEL
LIN {X 0,Y 608.544,Z 557.336,A -85,B 0,C 180,E1 -439.009,E2 -439.009} C_VEL
LIN {X 0,Y 608.506,Z 568.642,A -85,B 0,C 180,E1 -439.52,E2 -439.52} C_VEL
LIN {X 0,Y 608.48,Z 580.203,A -85,B 0,C 180,E1 -440.191,E2 -440.191} C_VEL
LIN {X 0,Y 608.485,Z 590.598,A -85,B 0,C 180,E1 -440.946,E2 -440.946} C_VEL
LIN {X 0,Y 608.475,Z 599.115,A -85,B 0,C 180,E1 -441.699,E2 -441.699} C_VEL
LIN {X 0,Y 608.471,Z 606.963,A -85,B 0,C 180,E1 -442.534,E2 -442.534} C_VEL
LIN {X 0,Y 608.46,Z 614.288,A -85,B 0,C 180,E1 -443.485,E2 -443.485} C_VEL
LIN {X 0,Y 608.45,Z 619.867,A -85,B 0,C 180,E1 -444.366,E2 -444.366} C_VEL
LIN {X 0,Y 608.432,Z 624.951,A -85,B 0,C 180,E1 -445.362,E2 -445.362} C_VEL
LIN {X 0,Y 608.449,Z 628.897,A -85,B 0,C 180,E1 -446.358,E2 -446.358} C_VEL
LIN {X 0,Y 608.425,Z 631.81,A -85,B 0,C 180,E1 -447.352,E2 -447.352} C_VEL
LIN {X 0,Y 608.442,Z 633.202,A -85,B 0,C 180,E1 -448.014,E2 -448.014} C_VEL
LIN {X 0,Y 608.438,Z 634.784,A -85,B 0,C 180,E1 -449.338,E2 -449.338} C_VEL
LIN {X 0,Y 608.434,Z 635,A -85,B 0,C 180,E1 -450,E2 -450} C_VEL
LIN {X 0,Y 608.448,Z 634.184,A -85,B 0,C 180,E1 -451.324,E2 -451.324} C_VEL
LIN {X 0,Y 608.443,Z 633.201,A -85,B 0,C 180,E1 -451.986,E2 -451.986} C_VEL
LIN {X 0,Y 608.425,Z 631.809,A -85,B 0,C 180,E1 -452.648,E2 -452.648} C_VEL
LIN {X 0,Y 608.449,Z 628.896,A -85,B 0,C 180,E1 -453.642,E2 -453.642} C_VEL
LIN {X 0,Y 608.432,Z 624.95,A -85,B 0,C 180,E1 -454.638,E2 -454.638} C_VEL
LIN {X 0,Y 608.437,Z 618.876,A -85,B 0,C 180,E1 -455.801,E2 -455.801} C_VEL
LIN {X 0,Y 608.462,Z 612.235,A -85,B 0,C 180,E1 -456.799,E2 -456.799} C_VEL
LIN {X 0,Y 608.456,Z 603.989,A -85,B 0,C 180,E1 -457.8,E2 -457.8} C_VEL
LIN {X 0,Y 608.472,Z 595.536,A -85,B 0,C 180,E1 -458.636,E2 -458.636} C_VEL
LIN {X 0,Y 608.471,Z 585.091,A -85,B 0,C 180,E1 -459.473,E2 -459.473} C_VEL
LIN {X 0,Y 608.495,Z 574.756,A -85,B 0,C 180,E1 -460.145,E2 -460.145} C_VEL
LIN {X 0,Y 608.522,Z 563.241,A -85,B 0,C 180,E1 -460.741,E2 -460.741} C_VEL
LIN {X 0,Y 608.533,Z 551.876,A -85,B 0,C 180,E1 -461.193,E2 -461.193} C_VEL
LIN {X 0,Y 608.562,Z 538.356,A -85,B 0,C 180,E1 -461.575,E2 -461.575} C_VEL
LIN {X 0,Y 608.555,Z 525.09,A -85,B 0,C 180,E1 -461.808,E2 -461.808} C_VEL
LIN {X 0,Y 608.558,Z 423.75,A -85,B 0,C 180,E1 -463.014,E2 -463.014} C_VEL
LIN {X 0,Y 608.485,Z 422.652,A -85,B 0,C 180,E1 -463.101,E2 -463.101} C_VEL
LIN {X 0,Y 608.495,Z 402.711,A -85,B 0,C 180,E1 -465.921,E2 -465.921} C_VEL
LIN {X 0,Y 608.514,Z 383.168,A -85,B 0,C 180,E1 -468.727,E2 -468.727} C_VEL
LIN {X 0,Y 608.571,Z 365.307,A -85,B 0,C 180,E1 -471.332,E2 -471.332} C_VEL
LIN {X 0,Y 608.488,Z 363.256,A -85,B 0,C 180,E1 -471.691,E2 -471.691} C_VEL
LIN {X 0,Y 608.452,Z 363.188,A -85,B 0,C 180,E1 -474.571,E2 -474.571} C_VEL
LIN {X 0,Y 608.483,Z 363.189,A -85,B 0,C 180,E1 -477.208,E2 -477.208} C_VEL
LIN {X 0,Y 608.472,Z 363.188,A -85,B 0,C 180,E1 -479.972,E2 -479.972} C_VEL
LIN {X 0,Y 608.456,Z 363.187,A -85,B 0,C 180,E1 -482.521,E2 -482.521} C_VEL
LIN {X 0,Y 608.453,Z 363.196,A -85,B 0,C 180,E1 -485.276,E2 -485.276} C_VEL
LIN {X 0,Y 608.47,Z 363.189,A -85,B 0,C 180,E1 -487.745,E2 -487.745} C_VEL
LIN {X 0,Y 608.445,Z 363.188,A -85,B 0,C 180,E1 -490.328,E2 -490.328} C_VEL
LIN {X 0,Y 608.485,Z 363.193,A -85,B 0,C 180,E1 -493.31,E2 -493.31} C_VEL
LIN {X 0,Y 608.469,Z 363.185,A -85,B 0,C 180,E1 -496.13,E2 -496.13} C_VEL
LIN {X 0,Y 608.461,Z 363.192,A -85,B 0,C 180,E1 -498.824,E2 -498.824} C_VEL
LIN {X 0,Y 608.467,Z 363.187,A -85,B 0,C 180,E1 -501.759,E2 -501.759} C_VEL
LIN {X 0,Y 608.473,Z 363.185,A -85,B 0,C 180,E1 -503.95,E2 -503.95} C_VEL
LIN {X 0,Y 608.461,Z 363.188,A -85,B 0,C 180,E1 -506.329,E2 -506.329} C_VEL
LIN {X 0,Y 608.473,Z 363.192,A -85,B 0,C 180,E1 -508.727,E2 -508.727} C_VEL
LIN {X 0,Y 608.471,Z 363.188,A -85,B 0,C 180,E1 -511.379,E2 -511.379} C_VEL
LIN {X 0,Y 608.445,Z 363.189,A -85,B 0,C 180,E1 -513.964,E2 -513.964} C_VEL
LIN {X 0,Y 608.46,Z 363.188,A -85,B 0,C 180,E1 -516.155,E2 -516.155} C_VEL
LIN {X 0,Y 608.471,Z 363.188,A -85,B 0,C 180,E1 -518.308,E2 -518.308} C_VEL
LIN {X 0,Y 608.467,Z 363.188,A -85,B 0,C 180,E1 -521.282,E2 -521.282} C_VEL
LIN {X 0,Y 608.456,Z 363.188,A -85,B 0,C 180,E1 -523.906,E2 -523.906} C_VEL
LIN {X 0,Y 608.46,Z 363.197,A -85,B 0,C 180,E1 -526.643,E2 -526.643} C_VEL
LIN {X 0,Y 608.465,Z 363.186,A -85,B 0,C 180,E1 -529.35,E2 -529.35} C_VEL
LIN {X 0,Y 608.47,Z 363.188,A -85,B 0,C 180,E1 -532.033,E2 -532.033} C_VEL
LIN {X 0,Y 608.462,Z 363.193,A -85,B 0,C 180,E1 -534.698,E2 -534.698} C_VEL
LIN {X 0,Y 608.479,Z 363.184,A -85,B 0,C 180,E1 -537.352,E2 -537.352} C_VEL
LIN {X 0,Y 608.469,Z 363.19,A -85,B 0,C 180,E1 -540,E2 -540} C_VEL
LIN {X 0,Y 608.479,Z 363.189,A -85,B 0,C 180,E1 -542.648,E2 -542.648} C_VEL
LIN {X 0,Y 608.463,Z 363.186,A -85,B 0,C 180,E1 -545.302,E2 -545.302} C_VEL
LIN {X 0,Y 608.473,Z 363.191,A -85,B 0,C 180,E1 -547.967,E2 -547.967} C_VEL
LIN {X 0,Y 608.452,Z 363.188,A -85,B 0,C 180,E1 -549.469,E2 -549.469} C_VEL
LIN {X 0,Y 607.774,Z 363.281,A -85,B 0,C 180,E1 -550.022,E2 -550.022} C_VEL
LIN {X 0,Y 604.918,Z 363.64,A -85,B 0,C 180,E1 -550.919,E2 -550.919} C_VEL
LIN {X 0,Y 602.516,Z 363.94,A -85,B 0,C 180,E1 -551.64,E2 -551.64} C_VEL
LIN {X 0,Y 601.488,Z 364.066,A -85,B 0,C 180,E1 -552.197,E2 -552.197} C_VEL
LIN {X 0,Y 601.406,Z 364.071,A -85,B 0,C 180,E1 -552.385,E2 -552.385} C_VEL
LIN {X 0,Y 601.43,Z 364.063,A -85,B 0,C 180,E1 -554.897,E2 -554.897} C_VEL
LIN {X 0,Y 601.43,Z 364.063,A -85,B 0,C 180,E1 -556.986,E2 -556.986} C_VEL
LIN {X 0,Y 601.408,Z 364.072,A -85,B 0,C 180,E1 -559.809,E2 -559.809} C_VEL
LIN {X 0,Y 601.408,Z 364.066,A -85,B 0,C 180,E1 -562.683,E2 -562.683} C_VEL
LIN {X 0,Y 601.401,Z 364.066,A -85,B 0,C 180,E1 -564.879,E2 -564.879} C_VEL
LIN {X 0,Y 601.422,Z 364.074,A -85,B 0,C 180,E1 -567.867,E2 -567.867} C_VEL
LIN {X 0,Y 601.444,Z 364.066,A -85,B 0,C 180,E1 -570.163,E2 -570.163} C_VEL
LIN {X 0,Y 601.423,Z 364.063,A -85,B 0,C 180,E1 -572.717,E2 -572.717} C_VEL
LIN {X 0,Y 601.407,Z 364.067,A -85,B 0,C 180,E1 -575.115,E2 -575.115} C_VEL
LIN {X 0,Y 601.433,Z 364.068,A -85,B 0,C 180,E1 -577.419,E2 -577.419} C_VEL
LIN {X 0,Y 601.41,Z 364.07,A -85,B 0,C 180,E1 -579.995,E2 -579.995} C_VEL
LIN {X 0,Y 601.412,Z 364.065,A -85,B 0,C 180,E1 -582.67,E2 -582.67} C_VEL
LIN {X 0,Y 601.423,Z 364.073,A -85,B 0,C 180,E1 -585.483,E2 -585.483} C_VEL
LIN {X 0,Y 601.422,Z 364.064,A -85,B 0,C 180,E1 -588.407,E2 -588.407} C_VEL
LIN {X 0,Y 601.434,Z 364.064,A -85,B 0,C 180,E1 -590.876,E2 -590.876} C_VEL
LIN {X 0,Y 601.443,Z 364.066,A -85,B 0,C 180,E1 -593.734,E2 -593.734} C_VEL
LIN {X 0,Y 601.432,Z 364.063,A -85,B 0,C 180,E1 -596.065,E2 -596.065} C_VEL
LIN {X 0,Y 601.43,Z 364.063,A -85,B 0,C 180,E1 -598.544,E2 -598.544} C_VEL
LIN {X 0,Y 601.434,Z 364.071,A -85,B 0,C 180,E1 -601.374,E2 -601.374} C_VEL
LIN {X 0,Y 601.412,Z 364.065,A -85,B 0,C 180,E1 -604.133,E2 -604.133} C_VEL
LIN {X 0,Y 601.419,Z 364.065,A -85,B 0,C 180,E1 -606.59,E2 -606.59} C_VEL
LIN {X 0,Y 601.429,Z 364.067,A -85,B 0,C 180,E1 -609.478,E2 -609.478} C_VEL
LIN {X 0,Y 601.398,Z 364.067,A -85,B 0,C 180,E1 -612.312,E2 -612.312} C_VEL
LIN {X 0,Y 601.413,Z 364.066,A -85,B 0,C 180,E1 -614.409,E2 -614.409} C_VEL
LIN {X 0,Y 601.416,Z 364.072,A -85,B 0,C 180,E1 -617.172,E2 -617.172} C_VEL
LIN {X 0,Y 601.436,Z 364.062,A -85,B 0,C 180,E1 -619.905,E2 -619.905} C_VEL
LIN {X 0,Y 601.453,Z 364.241,A -85,B 0,C 180,E1 -622.784,E2 -622.784} C_VEL
LIN {X 0,Y 601.535,Z 376.695,A -85,B 0,C 180,E1 -624.805,E2 -624.805} C_VEL
LIN {X 0,Y 601.485,Z 394.661,A -85,B 0,C 180,E1 -627.656,E2 -627.656} C_VEL
LIN {X 0,Y 601.437,Z 408.871,A -85,B 0,C 180,E1 -629.853,E2 -629.853} C_VEL
LIN {X 0,Y 601.659,Z 411.273,A -85,B 0,C 180,E1 -629.916,E2 -629.916} C_VEL
LIN {X 0,Y 601.606,Z 516.359,A -85,B 0,C 180,E1 -631.192,E2 -631.192} C_VEL
LIN {X 0,Y 601.579,Z 530.037,A -85,B 0,C 180,E1 -631.506,E2 -631.506} C_VEL
LIN {X 0,Y 601.535,Z 542.339,A -85,B 0,C 180,E1 -631.925,E2 -631.925} C_VEL
LIN {X 0,Y 601.525,Z 553.368,A -85,B 0,C 180,E1 -632.427,E2 -632.427} C_VEL
LIN {X 0,Y 601.479,Z 564.851,A -85,B 0,C 180,E1 -633.098,E2 -633.098} C_VEL
LIN {X 0,Y 601.452,Z 575.198,A -85,B 0,C 180,E1 -633.852,E2 -633.852} C_VEL
LIN {X 0,Y 601.417,Z 584.591,A -85,B 0,C 180,E1 -634.692,E2 -634.692} C_VEL
LIN {X 0,Y 601.391,Z 593.663,A -85,B 0,C 180,E1 -635.7,E2 -635.7} C_VEL
LIN {X 0,Y 601.381,Z 601.005,A -85,B 0,C 180,E1 -636.711,E2 -636.711} C_VEL
LIN {X 0,Y 601.354,Z 606.914,A -85,B 0,C 180,E1 -637.724,E2 -637.724} C_VEL
LIN {X 0,Y 601.347,Z 611.584,A -85,B 0,C 180,E1 -638.739,E2 -638.739} C_VEL
LIN {X 0,Y 601.34,Z 615.15,A -85,B 0,C 180,E1 -639.756,E2 -639.756} C_VEL
LIN {X 0,Y 601.351,Z 618.1,A -85,B 0,C 180,E1 -640.975,E2 -640.975} C_VEL
LIN {X 0,Y 601.342,Z 619.623,A -85,B 0,C 180,E1 -642.144,E2 -642.144} C_VEL
LIN {X 0,Y 601.34,Z 619.896,A -85,B 0,C 180,E1 -643.517,E2 -643.517} C_VEL
LIN {X 0,Y 601.319,Z 619.39,A -85,B 0,C 180,E1 -644.207,E2 -644.207} C_VEL
LIN {X 0,Y 601.314,Z 618.456,A -85,B 0,C 180,E1 -644.899,E2 -644.899} C_VEL
LIN {X 0,Y 601.325,Z 617.105,A -85,B 0,C 180,E1 -645.593,E2 -645.593} C_VEL
LIN {X 0,Y 601.326,Z 614.345,A -85,B 0,C 180,E1 -646.589,E2 -646.589} C_VEL
LIN {X 0,Y 601.347,Z 610.155,A -85,B 0,C 180,E1 -647.689,E2 -647.689} C_VEL
LIN {X 0,Y 601.382,Z 604.508,A -85,B 0,C 180,E1 -648.809,E2 -648.809} C_VEL
LIN {X 0,Y 601.372,Z 598.078,A -85,B 0,C 180,E1 -649.81,E2 -649.81} C_VEL
LIN {X 0,Y 601.411,Z 590.26,A -85,B 0,C 180,E1 -650.793,E2 -650.793} C_VEL
LIN {X 0,Y 601.429,Z 580.595,A -85,B 0,C 180,E1 -651.778,E2 -651.778} C_VEL
LIN {X 0,Y 601.455,Z 570.313,A -85,B 0,C 180,E1 -652.614,E2 -652.614} C_VEL
LIN {X 0,Y 601.485,Z 559.648,A -85,B 0,C 180,E1 -653.316,E2 -653.316} C_VEL
LIN {X 0,Y 601.539,Z 549.302,A -85,B 0,C 180,E1 -653.861,E2 -653.861} C_VEL
LIN {X 0,Y 601.579,Z 537.148,A -85,B 0,C 180,E1 -654.36,E2 -654.36} C_VEL
LIN {X 0,Y 601.596,Z 524.172,A -85,B 0,C 180,E1 -654.737,E2 -654.737} C_VEL
LIN {X 0,Y 601.622,Z 510.61,A -85,B 0,C 180,E1 -654.983,E2 -654.983} C_VEL
LIN {X 0,Y 601.577,Z 409.868,A -85,B 0,C 180,E1 -656.195,E2 -656.195} C_VEL
LIN {X 0,Y 601.426,Z 408.602,A -85,B 0,C 180,E1 -656.261,E2 -656.261} C_VEL
LIN {X 0,Y 601.474,Z 390.715,A -85,B 0,C 180,E1 -659.057,E2 -659.057} C_VEL
LIN {X 0,Y 601.536,Z 372.765,A -85,B 0,C 180,E1 -661.915,E2 -661.915} C_VEL
LIN {X 0,Y 601.467,Z 364.146,A -85,B 0,C 180,E1 -663.335,E2 -663.335} C_VEL
LIN {X 0,Y 601.441,Z 364.061,A -85,B 0,C 180,E1 -666.266,E2 -666.266} C_VEL
LIN {X 0,Y 601.44,Z 364.071,A -85,B 0,C 180,E1 -669.123,E2 -669.123} C_VEL
LIN {X 0,Y 601.422,Z 364.065,A -85,B 0,C 180,E1 -671.764,E2 -671.764} C_VEL
LIN {X 0,Y 601.419,Z 364.065,A -85,B 0,C 180,E1 -674.534,E2 -674.534} C_VEL
LIN {X 0,Y 601.437,Z 364.066,A -85,B 0,C 180,E1 -677.405,E2 -677.405} C_VEL
LIN {X 0,Y 601.41,Z 364.065,A -85,B 0,C 180,E1 -680.005,E2 -680.005} C_VEL
LIN {X 0,Y 601.433,Z 364.065,A -85,B 0,C 180,E1 -682.616,E2 -682.616} C_VEL
LIN {X 0,Y 601.438,Z 364.071,A -85,B 0,C 180,E1 -685.07,E2 -685.07} C_VEL
LIN {X 0,Y 601.432,Z 364.065,A -85,B 0,C 180,E1 -687.484,E2 -687.484} C_VEL
LIN {X 0,Y 601.44,Z 364.06,A -85,B 0,C 180,E1 -689.847,E2 -689.847} C_VEL
LIN {X 0,Y 601.419,Z 364.068,A -85,B 0,C 180,E1 -692.634,E2 -692.634} C_VEL
LIN {X 0,Y 601.404,Z 364.074,A -85,B 0,C 180,E1 -695.122,E2 -695.122} C_VEL
LIN {X 0,Y 601.45,Z 364.063,A -85,B 0,C 180,E1 -697.384,E2 -697.384} C_VEL
LIN {X 0,Y 601.406,Z 364.066,A -85,B 0,C 180,E1 -700.191,E2 -700.191} C_VEL
LIN {X 0,Y 601.43,Z 364.072,A -85,B 0,C 180,E1 -703.014,E2 -703.014} C_VEL
LIN {X 0,Y 601.412,Z 364.064,A -85,B 0,C 180,E1 -705.907,E2 -705.907} C_VEL
LIN {X 0,Y 601.431,Z 364.066,A -85,B 0,C 180,E1 -708.542,E2 -708.542} C_VEL
LIN {X 0,Y 601.438,Z 364.065,A -85,B 0,C 180,E1 -711.262,E2 -711.262} C_VEL
LIN {X 0,Y 601.404,Z 364.065,A -85,B 0,C 180,E1 -713.963,E2 -713.963} C_VEL
LIN {X 0,Y 601.438,Z 364.068,A -85,B 0,C 180,E1 -716.651,E2 -716.651} C_VEL
LIN {X 0,Y 601.451,Z 364.062,A -85,B 0,C 180,E1 -719.331,E2 -719.331} C_VEL
LIN {X 0,Y 601.418,Z 364.064,A -85,B 0,C 180,E1 -722.009,E2 -722.009} C_VEL
LIN {X 0,Y 601.432,Z 364.07,A -85,B 0,C 180,E1 -724.692,E2 -724.692} C_VEL
LIN {X 0,Y 601.448,Z 364.061,A -85,B 0,C 180,E1 -727.385,E2 -727.385} C_VEL
LIN {X 0,Y 601.43,Z 364.063,A -85,B 0,C 180,E1 -730.095,E2 -730.095} C_VEL
LIN {X 0,Y 601.425,Z 364.072,A -85,B 0,C 180,E1 -732.828,E2 -732.828} C_VEL
LIN {X 0,Y 601.414,Z 364.064,A -85,B 0,C 180,E1 -735.591,E2 -735.591} C_VEL
LIN {X 0,Y 601.419,Z 364.068,A -85,B 0,C 180,E1 -738.392,E2 -738.392} C_VEL
LIN {X 0,Y 601.408,Z 364.067,A -85,B 0,C 180,E1 -741.239,E2 -741.239} C_VEL
LIN {X 0,Y 601.418,Z 364.064,A -85,B 0,C 180,E1 -743.411,E2 -743.411} C_VEL
LIN {X 0,Y 601.404,Z 364.071,A -85,B 0,C 180,E1 -746.364,E2 -746.364} C_VEL
LIN {X 0,Y 601.442,Z 364.069,A -85,B 0,C 180,E1 -748.792,E2 -748.792} C_VEL
LIN {X 0,Y 601.412,Z 364.064,A -85,B 0,C 180,E1 -751.727,E2 -751.727} C_VEL
LIN {X 0,Y 601.427,Z 364.065,A -85,B 0,C 180,E1 -754.119,E2 -754.119} C_VEL
LIN {X 0,Y 601.412,Z 364.075,A -85,B 0,C 180,E1 -756.583,E2 -756.583} C_VEL
LIN {X 0,Y 601.434,Z 364.061,A -85,B 0,C 180,E1 -759.537,E2 -759.537} C_VEL
LIN {X 0,Y 601.437,Z 364.072,A -85,B 0,C 180,E1 -762.595,E2 -762.595} C_VEL
LIN {X 0,Y 601.421,Z 364.063,A -85,B 0,C 180,E1 -765.483,E2 -765.483} C_VEL
LIN {X 0,Y 601.425,Z 364.072,A -85,B 0,C 180,E1 -768.407,E2 -768.407} C_VEL
LIN {X 0,Y 601.437,Z 364.066,A -85,B 0,C 180,E1 -770.877,E2 -770.877} C_VEL
LIN {X 0,Y 601.442,Z 364.061,A -85,B 0,C 180,E1 -773.735,E2 -773.735} C_VEL
LIN {X 0,Y 601.436,Z 364.065,A -85,B 0,C 180,E1 -776.064,E2 -776.064} C_VEL
LIN {X 0,Y 601.431,Z 364.064,A -85,B 0,C 180,E1 -779.06,E2 -779.06} C_VEL
LIN {X 0,Y 601.429,Z 364.062,A -85,B 0,C 180,E1 -781.374,E2 -781.374} C_VEL
LIN {X 0,Y 601.404,Z 364.066,A -85,B 0,C 180,E1 -783.637,E2 -783.637} C_VEL
LIN {X 0,Y 601.423,Z 364.072,A -85,B 0,C 180,E1 -786.591,E2 -786.591} C_VEL
LIN {X 0,Y 601.463,Z 364.244,A -85,B 0,C 180,E1 -788.224,E2 -788.224} C_VEL
LIN {X 0,Y 601.605,Z 371.099,A -85,B 0,C 180,E1 -789.27,E2 -789.27} C_VEL
LIN {X 0,Y 601.536,Z 389.441,A -85,B 0,C 180,E1 -791.965,E2 -791.965} C_VEL
LIN {X 0,Y 601.455,Z 408.746,A -85,B 0,C 180,E1 -794.758,E2 -794.758} C_VEL
LIN {X 0,Y 601.469,Z 423.293,A -85,B 0,C 180,E1 -796.808,E2 -796.808} C_VEL
LIN {X 0,Y 601.687,Z 426.756,A -85,B 0,C 180,E1 -796.878,E2 -796.878} C_VEL
LIN {X 0,Y 601.623,Z 530.969,A -85,B 0,C 180,E1 -798.14,E2 -798.14} C_VEL
LIN {X 0,Y 601.59,Z 544.232,A -85,B 0,C 180,E1 -798.439,E2 -798.439} C_VEL
LIN {X 0,Y 601.575,Z 556.664,A -85,B 0,C 180,E1 -798.855,E2 -798.855} C_VEL
LIN {X 0,Y 601.527,Z 568.641,A -85,B 0,C 180,E1 -799.397,E2 -799.397} C_VEL
LIN {X 0,Y 601.48,Z 580.204,A -85,B 0,C 180,E1 -800.076,E2 -800.076} C_VEL
LIN {X 0,Y 601.444,Z 590.599,A -85,B 0,C 180,E1 -800.839,E2 -800.839} C_VEL
LIN {X 0,Y 601.429,Z 599.115,A -85,B 0,C 180,E1 -801.601,E2 -801.601} C_VEL
LIN {X 0,Y 601.418,Z 606.963,A -85,B 0,C 180,E1 -802.446,E2 -802.446} C_VEL
LIN {X 0,Y 601.37,Z 614.226,A -85,B 0,C 180,E1 -803.398,E2 -803.398} C_VEL
LIN {X 0,Y 601.372,Z 619.868,A -85,B 0,C 180,E1 -804.299,E2 -804.299} C_VEL
LIN {X 0,Y 601.337,Z 624.951,A -85,B 0,C 180,E1 -805.308,E2 -805.308} C_VEL
LIN {X 0,Y 601.367,Z 628.897,A -85,B 0,C 180,E1 -806.315,E2 -806.315} C_VEL
LIN {X 0,Y 601.325,Z 631.809,A -85,B 0,C 180,E1 -807.321,E2 -807.321} C_VEL
LIN {X 0,Y 601.341,Z 633.202,A -85,B 0,C 180,E1 -807.991,E2 -807.991} C_VEL
LIN {X 0,Y 601.339,Z 634.784,A -85,B 0,C 180,E1 -809.331,E2 -809.331} C_VEL
LIN {X 0,Y 601.335,Z 635,A -85,B 0,C 180,E1 -810,E2 -810} C_VEL
LIN {X 0,Y 601.348,Z 634.184,A -85,B 0,C 180,E1 -811.34,E2 -811.34} C_VEL
LIN {X 0,Y 601.341,Z 633.202,A -85,B 0,C 180,E1 -812.009,E2 -812.009} C_VEL
LIN {X 0,Y 601.325,Z 631.809,A -85,B 0,C 180,E1 -812.68,E2 -812.68} C_VEL
LIN {X 0,Y 601.367,Z 628.896,A -85,B 0,C 180,E1 -813.685,E2 -813.685} C_VEL
LIN {X 0,Y 601.337,Z 624.949,A -85,B 0,C 180,E1 -814.693,E2 -814.693} C_VEL
LIN {X 0,Y 601.372,Z 618.877,A -85,B 0,C 180,E1 -815.869,E2 -815.869} C_VEL
LIN {X 0,Y 601.382,Z 612.235,A -85,B 0,C 180,E1 -816.88,E2 -816.88} C_VEL
LIN {X 0,Y 601.4,Z 603.989,A -85,B 0,C 180,E1 -817.892,E2 -817.892} C_VEL
LIN {X 0,Y 601.436,Z 595.537,A -85,B 0,C 180,E1 -818.738,E2 -818.738} C_VEL
LIN {X 0,Y 601.442,Z 585.093,A -85,B 0,C 180,E1 -819.585,E2 -819.585} C_VEL
LIN {X 0,Y 601.472,Z 574.758,A -85,B 0,C 180,E1 -820.264,E2 -820.264} C_VEL
LIN {X 0,Y 601.537,Z 563.897,A -85,B 0,C 180,E1 -820.836,E2 -820.836} C_VEL
LIN {X 0,Y 601.565,Z 551.375,A -85,B 0,C 180,E1 -821.34,E2 -821.34} C_VEL
LIN {X 0,Y 601.607,Z 538.355,A -85,B 0,C 180,E1 -821.711,E2 -821.711} C_VEL
LIN {X 0,Y 601.625,Z 525.09,A -85,B 0,C 180,E1 -821.946,E2 -821.946} C_VEL
LIN {X 0,Y 601.527,Z 423.736,A -85,B 0,C 180,E1 -823.169,E2 -823.169} C_VEL
LIN {X 0,Y 601.464,Z 422.652,A -85,B 0,C 180,E1 -823.257,E2 -823.257} C_VEL
LIN {X 0,Y 601.511,Z 401.504,A -85,B 0,C 180,E1 -826.285,E2 -826.285} C_VEL
LIN {X 0,Y 601.574,Z 380.992,A -85,B 0,C 180,E1 -829.271,E2 -829.271} C_VEL
LIN {X 0,Y 601.539,Z 364.703,A -85,B 0,C 180,E1 -831.684,E2 -831.684} C_VEL
LIN {X 0,Y 601.426,Z 364.094,A -85,B 0,C 180,E1 -831.868,E2 -831.868} C_VEL
LIN {X 0,Y 601.435,Z 364.063,A -85,B 0,C 180,E1 -834.292,E2 -834.292} C_VEL
LIN {X 0,Y 601.455,Z 364.063,A -85,B 0,C 180,E1 -837.111,E2 -837.111} C_VEL
LIN {X 0,Y 601.428,Z 364.072,A -85,B 0,C 180,E1 -839.392,E2 -839.392} C_VEL
LIN {X 0,Y 601.414,Z 364.07,A -85,B 0,C 180,E1 -841.726,E2 -841.726} C_VEL
LIN {X 0,Y 601.432,Z 364.063,A -85,B 0,C 180,E1 -844.118,E2 -844.118} C_VEL
LIN {X 0,Y 601.415,Z 364.065,A -85,B 0,C 180,E1 -846.581,E2 -846.581} C_VEL
LIN {X 0,Y 601.444,Z 364.067,A -85,B 0,C 180,E1 -849.536,E2 -849.536} C_VEL
LIN {X 0,Y 601.423,Z 364.066,A -85,B 0,C 180,E1 -851.764,E2 -851.764} C_VEL
LIN {X 0,Y 601.422,Z 364.065,A -85,B 0,C 180,E1 -854.535,E2 -854.535} C_VEL
LIN {X 0,Y 601.438,Z 364.067,A -85,B 0,C 180,E1 -857.406,E2 -857.406} C_VEL
LIN {X 0,Y 601.411,Z 364.065,A -85,B 0,C 180,E1 -860.005,E2 -860.005} C_VEL
LIN {X 0,Y 601.435,Z 364.065,A -85,B 0,C 180,E1 -862.617,E2 -862.617} C_VEL
LIN {X 0,Y 601.437,Z 364.071,A -85,B 0,C 180,E1 -865.069,E2 -865.069} C_VEL
LIN {X 0,Y 601.432,Z 364.065,A -85,B 0,C 180,E1 -867.484,E2 -867.484} C_VEL
LIN {X 0,Y 601.423,Z 364.063,A -85,B 0,C 180,E1 -869.851,E2 -869.851} C_VEL
LIN {X 0,Y 601.417,Z 364.07,A -85,B 0,C 180,E1 -872.636,E2 -872.636} C_VEL
LIN {X 0,Y 601.4,Z 364.072,A -85,B 0,C 180,E1 -875.121,E2 -875.121} C_VEL
LIN {X 0,Y 601.41,Z 364.067,A -85,B 0,C 180,E1 -877.394,E2 -877.394} C_VEL
LIN {X 0,Y 601.405,Z 364.068,A -85,B 0,C 180,E1 -880.19,E2 -880.19} C_VEL
LIN {X 0,Y 601.431,Z 364.067,A -85,B 0,C 180,E1 -883.014,E2 -883.014} C_VEL
LIN {X 0,Y 601.414,Z 364.065,A -85,B 0,C 180,E1 -885.907,E2 -885.907} C_VEL
LIN {X 0,Y 601.429,Z 364.073,A -85,B 0,C 180,E1 -888.542,E2 -888.542} C_VEL
LIN {X 0,Y 601.434,Z 364.063,A -85,B 0,C 180,E1 -891.262,E2 -891.262} C_VEL
LIN {X 0,Y 601.405,Z 364.068,A -85,B 0,C 180,E1 -893.963,E2 -893.963} C_VEL
LIN {X 0,Y 601.428,Z 364.07,A -85,B 0,C 180,E1 -896.65,E2 -896.65} C_VEL
LIN {X 0,Y 601.447,Z 364.06,A -85,B 0,C 180,E1 -899.33,E2 -899.33} C_VEL
LIN {X 0,Y 601.42,Z 364.069,A -85,B 0,C 180,E1 -902.009,E2 -902.009} C_VEL
LIN {X 0,Y 601.426,Z 364.067,A -85,B 0,C 180,E1 -904.692,E2 -904.692} C_VEL
LIN {X 0,Y 601.447,Z 364.061,A -85,B 0,C 180,E1 -907.385,E2 -907.385} C_VEL
LIN {X 0,Y 601.429,Z 364.071,A -85,B 0,C 180,E1 -910.095,E2 -910.095} C_VEL
LIN {X 0,Y 601.406,Z 364.071,A -85,B 0,C 180,E1 -912.385,E2 -912.385} C_VEL
LIN {X 0,Y 600.743,Z 364.15,A -85,B 0,C 180,E1 -912.945,E2 -912.945} C_VEL
LIN {X 0,Y 597.893,Z 364.509,A -85,B 0,C 180,E1 -913.853,E2 -913.853} C_VEL
LIN {X 0,Y 595.483,Z 364.807,A -85,B 0,C 180,E1 -914.583,E2 -914.583} C_VEL
LIN {X 0,Y 594.449,Z 364.933,A -85,B 0,C 180,E1 -915.146,E2 -915.146} C_VEL
LIN {X 0,Y 594.365,Z 364.943,A -85,B 0,C 180,E1 -915.337,E2 -915.337} C_VEL
LIN {X 0,Y 594.38,Z 364.949,A -85,B 0,C 180,E1 -917.904,E2 -917.904} C_VEL
LIN {X 0,Y 594.377,Z 364.941,A -85,B 0,C 180,E1 -920.918,E2 -920.918} C_VEL
LIN {X 0,Y 594.393,Z 364.945,A -85,B 0,C 180,E1 -923.704,E2 -923.704} C_VEL
LIN {X 0,Y 594.383,Z 364.941,A -85,B 0,C 180,E1 -926.7,E2 -926.7} C_VEL
LIN {X 0,Y 594.38,Z 364.941,A -85,B 0,C 180,E1 -928.999,E2 -928.999} C_VEL
LIN {X 0,Y 594.392,Z 364.947,A -85,B 0,C 180,E1 -931.646,E2 -931.646} C_VEL
LIN {X 0,Y 594.389,Z 364.94,A -85,B 0,C 180,E1 -934.579,E2 -934.579} C_VEL
LIN {X 0,Y 594.383,Z 364.942,A -85,B 0,C 180,E1 -937.087,E2 -937.087} C_VEL
LIN {X 0,Y 594.375,Z 364.95,A -85,B 0,C 180,E1 -939.775,E2 -939.775} C_VEL
LIN {X 0,Y 594.37,Z 364.943,A -85,B 0,C 180,E1 -942.375,E2 -942.375} C_VEL
LIN {X 0,Y 594.36,Z 364.948,A -85,B 0,C 180,E1 -945.192,E2 -945.192} C_VEL
LIN {X 0,Y 594.382,Z 364.942,A -85,B 0,C 180,E1 -948.152,E2 -948.152} C_VEL
LIN {X 0,Y 594.392,Z 364.939,A -85,B 0,C 180,E1 -950.322,E2 -950.322} C_VEL
LIN {X 0,Y 594.384,Z 364.943,A -85,B 0,C 180,E1 -952.914,E2 -952.914} C_VEL
LIN {X 0,Y 594.386,Z 364.943,A -85,B 0,C 180,E1 -955.861,E2 -955.861} C_VEL
LIN {X 0,Y 594.379,Z 364.942,A -85,B 0,C 180,E1 -958.651,E2 -958.651} C_VEL
LIN {X 0,Y 594.384,Z 364.946,A -85,B 0,C 180,E1 -961.042,E2 -961.042} C_VEL
LIN {X 0,Y 594.387,Z 364.94,A -85,B 0,C 180,E1 -963.977,E2 -963.977} C_VEL
LIN {X 0,Y 594.389,Z 364.94,A -85,B 0,C 180,E1 -966.296,E2 -966.296} C_VEL
LIN {X 0,Y 594.403,Z 364.947,A -85,B 0,C 180,E1 -969.225,E2 -969.225} C_VEL
LIN {X 0,Y 594.356,Z 364.944,A -85,B 0,C 180,E1 -972.095,E2 -972.095} C_VEL
LIN {X 0,Y 594.366,Z 364.943,A -85,B 0,C 180,E1 -974.219,E2 -974.219} C_VEL
LIN {X 0,Y 594.384,Z 364.941,A -85,B 0,C 180,E1 -976.321,E2 -976.321} C_VEL
LIN {X 0,Y 594.377,Z 364.95,A -85,B 0,C 180,E1 -979.095,E2 -979.095} C_VEL
LIN {X 0,Y 594.415,Z 364.94,A -85,B 0,C 180,E1 -981.843,E2 -981.843} C_VEL
LIN {X 0,Y 594.424,Z 365.105,A -85,B 0,C 180,E1 -982.677,E2 -982.677} C_VEL
LIN {X 0,Y 594.536,Z 374.543,A -85,B 0,C 180,E1 -984.233,E2 -984.233} C_VEL
LIN {X 0,Y 594.465,Z 390.352,A -85,B 0,C 180,E1 -986.781,E2 -986.781} C_VEL
LIN {X 0,Y 594.41,Z 408.526,A -85,B 0,C 180,E1 -989.661,E2 -989.661} C_VEL
LIN {X 0,Y 594.52,Z 409.808,A -85,B 0,C 180,E1 -989.735,E2 -989.735} C_VEL
LIN {X 0,Y 594.754,Z 422.223,A -85,B 0,C 180,E1 -989.894,E2 -989.894} C_VEL
LIN {X 0,Y 594.669,Z 516.679,A -85,B 0,C 180,E1 -991.058,E2 -991.058} C_VEL
LIN {X 0,Y 594.637,Z 530.248,A -85,B 0,C 180,E1 -991.375,E2 -991.375} C_VEL
LIN {X 0,Y 594.55,Z 543.035,A -85,B 0,C 180,E1 -991.82,E2 -991.82} C_VEL
LIN {X 0,Y 594.531,Z 554.662,A -85,B 0,C 180,E1 -992.371,E2 -992.371} C_VEL
LIN {X 0,Y 594.468,Z 565.897,A -85,B 0,C 180,E1 -993.049,E2 -993.049} C_VEL
LIN {X 0,Y 594.417,Z 576.071,A -85,B 0,C 180,E1 -993.813,E2 -993.813} C_VEL
LIN {X 0,Y 594.384,Z 584.442,A -85,B 0,C 180,E1 -994.577,E2 -994.577} C_VEL
LIN {X 0,Y 594.314,Z 593.551,A -85,B 0,C 180,E1 -995.598,E2 -995.598} C_VEL
LIN {X 0,Y 594.29,Z 600.77,A -85,B 0,C 180,E1 -996.599,E2 -996.599} C_VEL
LIN {X 0,Y 594.28,Z 605.924,A -85,B 0,C 180,E1 -997.474,E2 -997.474} C_VEL
LIN {X 0,Y 594.285,Z 610.803,A -85,B 0,C 180,E1 -998.501,E2 -998.501} C_VEL
LIN {X 0,Y 594.266,Z 614.567,A -85,B 0,C 180,E1 -999.53,E2 -999.53} C_VEL
LIN {X 0,Y 594.233,Z 616.511,A -85,B 0,C 180,E1 -1000.218,E2 -1000.218} C_VEL
LIN {X 0,Y 594.263,Z 618.199,A -85,B 0,C 180,E1 -1001.01,E2 -1001.01} C_VEL
LIN {X 0,Y 594.239,Z 619.732,A -85,B 0,C 180,E1 -1002.291,E2 -1002.291} C_VEL
LIN {X 0,Y 594.243,Z 619.992,A -85,B 0,C 180,E1 -1002.985,E2 -1002.985} C_VEL
LIN {X 0,Y 594.26,Z 619.498,A -85,B 0,C 180,E1 -1004.124,E2 -1004.124} C_VEL
LIN {X 0,Y 594.209,Z 618.196,A -85,B 0,C 180,E1 -1005.082,E2 -1005.082} C_VEL
LIN {X 0,Y 594.252,Z 616.74,A -85,B 0,C 180,E1 -1005.784,E2 -1005.784} C_VEL
LIN {X 0,Y 594.24,Z 614.228,A -85,B 0,C 180,E1 -1006.669,E2 -1006.669} C_VEL
LIN {X 0,Y 594.263,Z 609.44,A -85,B 0,C 180,E1 -1007.907,E2 -1007.907} C_VEL
LIN {X 0,Y 594.321,Z 603.299,A -85,B 0,C 180,E1 -1009.081,E2 -1009.081} C_VEL
LIN {X 0,Y 594.314,Z 595.574,A -85,B 0,C 180,E1 -1010.236,E2 -1010.236} C_VEL
LIN {X 0,Y 594.386,Z 587.765,A -85,B 0,C 180,E1 -1011.165,E2 -1011.165} C_VEL
LIN {X 0,Y 594.423,Z 577.682,A -85,B 0,C 180,E1 -1012.139,E2 -1012.139} C_VEL
LIN {X 0,Y 594.442,Z 567.051,A -85,B 0,C 180,E1 -1012.963,E2 -1012.963} C_VEL
LIN {X 0,Y 594.501,Z 555.043,A -85,B 0,C 180,E1 -1013.699,E2 -1013.699} C_VEL
LIN {X 0,Y 594.565,Z 543.448,A -85,B 0,C 180,E1 -1014.252,E2 -1014.252} C_VEL
LIN {X 0,Y 594.637,Z 531.113,A -85,B 0,C 180,E1 -1014.69,E2 -1014.69} C_VEL
LIN {X 0,Y 594.672,Z 517.569,A -85,B 0,C 180,E1 -1015.015,E2 -1015.015} C_VEL
LIN {X 0,Y 594.698,Z 488.915,A -85,B 0,C 180,E1 -1015.388,E2 -1015.388} C_VEL
LIN {X 0,Y 594.649,Z 410.611,A -85,B 0,C 180,E1 -1016.339,E2 -1016.339} C_VEL
LIN {X 0,Y 594.391,Z 408.877,A -85,B 0,C 180,E1 -1016.395,E2 -1016.395} C_VEL
LIN {X 0,Y 594.457,Z 392.325,A -85,B 0,C 180,E1 -1018.994,E2 -1018.994} C_VEL
LIN {X 0,Y 594.554,Z 374.501,A -85,B 0,C 180,E1 -1021.863,E2 -1021.863} C_VEL
LIN {X 0,Y 594.438,Z 365.182,A -85,B 0,C 180,E1 -1023.4,E2 -1023.4} C_VEL
LIN {X 0,Y 594.385,Z 364.944,A -85,B 0,C 180,E1 -1024.139,E2 -1024.139} C_VEL
LIN {X 0,Y 594.386,Z 364.95,A -85,B 0,C 180,E1 -1027.086,E2 -1027.086} C_VEL
LIN {X 0,Y 594.376,Z 364.943,A -85,B 0,C 180,E1 -1029.774,E2 -1029.774} C_VEL
LIN {X 0,Y 594.365,Z 364.943,A -85,B 0,C 180,E1 -1032.374,E2 -1032.374} C_VEL
LIN {X 0,Y 594.358,Z 364.953,A -85,B 0,C 180,E1 -1035.19,E2 -1035.19} C_VEL
LIN {X 0,Y 594.385,Z 364.942,A -85,B 0,C 180,E1 -1037.626,E2 -1037.626} C_VEL
LIN {X 0,Y 594.388,Z 364.94,A -85,B 0,C 180,E1 -1040.321,E2 -1040.321} C_VEL
LIN {X 0,Y 594.384,Z 364.948,A -85,B 0,C 180,E1 -1042.913,E2 -1042.913} C_VEL
LIN {X 0,Y 594.38,Z 364.94,A -85,B 0,C 180,E1 -1045.86,E2 -1045.86} C_VEL
LIN {X 0,Y 594.386,Z 364.944,A -85,B 0,C 180,E1 -1048.651,E2 -1048.651} C_VEL
LIN {X 0,Y 594.383,Z 364.95,A -85,B 0,C 180,E1 -1051.04,E2 -1051.04} C_VEL
LIN {X 0,Y 594.384,Z 364.94,A -85,B 0,C 180,E1 -1053.975,E2 -1053.975} C_VEL
LIN {X 0,Y 594.385,Z 364.941,A -85,B 0,C 180,E1 -1056.296,E2 -1056.296} C_VEL
LIN {X 0,Y 594.404,Z 364.944,A -85,B 0,C 180,E1 -1059.224,E2 -1059.224} C_VEL
LIN {X 0,Y 594.377,Z 364.941,A -85,B 0,C 180,E1 -1062.096,E2 -1062.096} C_VEL
LIN {X 0,Y 594.368,Z 364.943,A -85,B 0,C 180,E1 -1064.219,E2 -1064.219} C_VEL
LIN {X 0,Y 594.371,Z 364.95,A -85,B 0,C 180,E1 -1067.017,E2 -1067.017} C_VEL
LIN {X 0,Y 594.391,Z 364.939,A -85,B 0,C 180,E1 -1069.784,E2 -1069.784} C_VEL
LIN {X 0,Y 594.413,Z 364.941,A -85,B 0,C 180,E1 -1072.527,E2 -1072.527} C_VEL
LIN {X 0,Y 594.396,Z 364.942,A -85,B 0,C 180,E1 -1075.252,E2 -1075.252} C_VEL
LIN {X 0,Y 594.389,Z 364.939,A -85,B 0,C 180,E1 -1077.967,E2 -1077.967} C_VEL
LIN {X 0,Y 594.427,Z 364.942,A -85,B 0,C 180,E1 -1080.677,E2 -1080.677} C_VEL
LIN {X 0,Y 594.384,Z 364.941,A -85,B 0,C 180,E1 -1083.389,E2 -1083.389} C_VEL
LIN {X 0,Y 594.361,Z 364.944,A -85,B 0,C 180,E1 -1086.109,E2 -1086.109} C_VEL
LIN {X 0,Y 594.411,Z 364.938,A -85,B 0,C 180,E1 -1088.157,E2 -1088.157} C_VEL
LIN {X 0,Y 594.391,Z 364.944,A -85,B 0,C 180,E1 -1091.081,E2 -1091.081} C_VEL
LIN {X 0,Y 594.377,Z 364.94,A -85,B 0,C 180,E1 -1093.679,E2 -1093.679} C_VEL
LIN {X 0,Y 594.394,Z 364.949,A -85,B 0,C 180,E1 -1096.723,E2 -1096.723} C_VEL
LIN {X 0,Y 594.364,Z 364.944,A -85,B 0,C 180,E1 -1099.335,E2 -1099.335} C_VEL
LIN {X 0,Y 594.366,Z 364.942,A -85,B 0,C 180,E1 -1101.503,E2 -1101.503} C_VEL
LIN {X 0,Y 594.386,Z 364.939,A -85,B 0,C 180,E1 -1103.704,E2 -1103.704} C_VEL
LIN {X 0,Y 594.384,Z 364.95,A -85,B 0,C 180,E1 -1106.7,E2 -1106.7} C_VEL
LIN {X 0,Y 594.381,Z 364.945,A -85,B 0,C 180,E1 -1108.999,E2 -1108.999} C_VEL
LIN {X 0,Y 594.388,Z 364.939,A -85,B 0,C 180,E1 -1111.646,E2 -1111.646} C_VEL
LIN {X 0,Y 594.392,Z 364.949,A -85,B 0,C 180,E1 -1114.579,E2 -1114.579} C_VEL
LIN {X 0,Y 594.383,Z 364.943,A -85,B 0,C 180,E1 -1117.087,E2 -1117.087} C_VEL
LIN {X 0,Y 594.372,Z 364.942,A -85,B 0,C 180,E1 -1119.776,E2 -1119.776} C_VEL
LIN {X 0,Y 594.385,Z 364.946,A -85,B 0,C 180,E1 -1122.374,E2 -1122.374} C_VEL
LIN {X 0,Y 594.358,Z 364.944,A -85,B 0,C 180,E1 -1125.192,E2 -1125.192} C_VEL
LIN {X 0,Y 594.365,Z 364.942,A -85,B 0,C 180,E1 -1127.626,E2 -1127.626} C_VEL
LIN {X 0,Y 594.392,Z 364.946,A -85,B 0,C 180,E1 -1130.322,E2 -1130.322} C_VEL
LIN {X 0,Y 594.385,Z 364.943,A -85,B 0,C 180,E1 -1132.914,E2 -1132.914} C_VEL
LIN {X 0,Y 594.386,Z 364.941,A -85,B 0,C 180,E1 -1135.861,E2 -1135.861} C_VEL
LIN {X 0,Y 594.391,Z 364.946,A -85,B 0,C 180,E1 -1138.652,E2 -1138.652} C_VEL
LIN {X 0,Y 594.383,Z 364.942,A -85,B 0,C 180,E1 -1141.043,E2 -1141.043} C_VEL
LIN {X 0,Y 594.392,Z 364.943,A -85,B 0,C 180,E1 -1143.977,E2 -1143.977} C_VEL
LIN {X 0,Y 594.391,Z 364.949,A -85,B 0,C 180,E1 -1146.297,E2 -1146.297} C_VEL
LIN {X 0,Y 594.407,Z 365.137,A -85,B 0,C 180,E1 -1148.089,E2 -1148.089} C_VEL
LIN {X 0,Y 594.692,Z 368.845,A -85,B 0,C 180,E1 -1148.679,E2 -1148.679} C_VEL
LIN {X 0,Y 594.57,Z 388.234,A -85,B 0,C 180,E1 -1151.568,E2 -1151.568} C_VEL
LIN {X 0,Y 594.487,Z 406.333,A -85,B 0,C 180,E1 -1154.223,E2 -1154.223} C_VEL
LIN {X 0,Y 594.436,Z 423.287,A -85,B 0,C 180,E1 -1156.649,E2 -1156.649} C_VEL
LIN {X 0,Y 594.774,Z 426.756,A -85,B 0,C 180,E1 -1156.722,E2 -1156.722} C_VEL
LIN {X 0,Y 594.692,Z 530.969,A -85,B 0,C 180,E1 -1158,E2 -1158} C_VEL
LIN {X 0,Y 594.639,Z 544.232,A -85,B 0,C 180,E1 -1158.302,E2 -1158.302} C_VEL
LIN {X 0,Y 594.591,Z 557.376,A -85,B 0,C 180,E1 -1158.749,E2 -1158.749} C_VEL
LIN {X 0,Y 594.539,Z 568.64,A -85,B 0,C 180,E1 -1159.27,E2 -1159.27} C_VEL
LIN {X 0,Y 594.477,Z 580.206,A -85,B 0,C 180,E1 -1159.958,E2 -1159.958} C_VEL
LIN {X 0,Y 594.413,Z 590.601,A -85,B 0,C 180,E1 -1160.73,E2 -1160.73} C_VEL
LIN {X 0,Y 594.383,Z 599.116,A -85,B 0,C 180,E1 -1161.501,E2 -1161.501} C_VEL
LIN {X 0,Y 594.347,Z 606.963,A -85,B 0,C 180,E1 -1162.356,E2 -1162.356} C_VEL
LIN {X 0,Y 594.282,Z 614.814,A -85,B 0,C 180,E1 -1163.409,E2 -1163.409} C_VEL
LIN {X 0,Y 594.289,Z 621.682,A -85,B 0,C 180,E1 -1164.572,E2 -1164.572} C_VEL
LIN {X 0,Y 594.27,Z 626.372,A -85,B 0,C 180,E1 -1165.592,E2 -1165.592} C_VEL
LIN {X 0,Y 594.267,Z 629.957,A -85,B 0,C 180,E1 -1166.61,E2 -1166.61} C_VEL
LIN {X 0,Y 594.226,Z 631.809,A -85,B 0,C 180,E1 -1167.289,E2 -1167.289} C_VEL
LIN {X 0,Y 594.24,Z 633.202,A -85,B 0,C 180,E1 -1167.967,E2 -1167.967} C_VEL
LIN {X 0,Y 594.239,Z 634.784,A -85,B 0,C 180,E1 -1169.323,E2 -1169.323} C_VEL
LIN {X 0,Y 594.236,Z 635,A -85,B 0,C 180,E1 -1170,E2 -1170} C_VEL
LIN {X 0,Y 594.247,Z 634.185,A -85,B 0,C 180,E1 -1171.356,E2 -1171.356} C_VEL
LIN {X 0,Y 594.24,Z 633.201,A -85,B 0,C 180,E1 -1172.033,E2 -1172.033} C_VEL
LIN {X 0,Y 594.226,Z 631.809,A -85,B 0,C 180,E1 -1172.712,E2 -1172.712} C_VEL
LIN {X 0,Y 594.288,Z 628.896,A -85,B 0,C 180,E1 -1173.729,E2 -1173.729} C_VEL
LIN {X 0,Y 594.242,Z 624.949,A -85,B 0,C 180,E1 -1174.749,E2 -1174.749} C_VEL
LIN {X 0,Y 594.304,Z 618.877,A -85,B 0,C 180,E1 -1175.939,E2 -1175.939} C_VEL
LIN {X 0,Y 594.308,Z 612.236,A -85,B 0,C 180,E1 -1176.962,E2 -1176.962} C_VEL
LIN {X 0,Y 594.359,Z 603.99,A -85,B 0,C 180,E1 -1177.986,E2 -1177.986} C_VEL
LIN {X 0,Y 594.382,Z 595.537,A -85,B 0,C 180,E1 -1178.842,E2 -1178.842} C_VEL
LIN {X 0,Y 594.427,Z 585.094,A -85,B 0,C 180,E1 -1179.699,E2 -1179.699} C_VEL
LIN {X 0,Y 594.486,Z 574.76,A -85,B 0,C 180,E1 -1180.386,E2 -1180.386} C_VEL
LIN {X 0,Y 594.561,Z 563.692,A -85,B 0,C 180,E1 -1180.975,E2 -1180.975} C_VEL
LIN {X 0,Y 594.6,Z 551.703,A -85,B 0,C 180,E1 -1181.464,E2 -1181.464} C_VEL
LIN {X 0,Y 594.656,Z 538.354,A -85,B 0,C 180,E1 -1181.85,E2 -1181.85} C_VEL
LIN {X 0,Y 594.697,Z 525.09,A -85,B 0,C 180,E1 -1182.087,E2 -1182.087} C_VEL
LIN {X 0,Y 594.612,Z 424.518,A -85,B 0,C 180,E1 -1183.309,E2 -1183.309} C_VEL
LIN {X 0,Y 594.43,Z 423.005,A -85,B 0,C 180,E1 -1183.373,E2 -1183.373} C_VEL
LIN {X 0,Y 594.501,Z 403.918,A -85,B 0,C 180,E1 -1186.129,E2 -1186.129} C_VEL
LIN {X 0,Y 594.593,Z 385.252,A -85,B 0,C 180,E1 -1188.873,E2 -1188.873} C_VEL
LIN {X 0,Y 594.7,Z 367.72,A -85,B 0,C 180,E1 -1191.49,E2 -1191.49} C_VEL
LIN {X 0,Y 594.393,Z 364.994,A -85,B 0,C 180,E1 -1191.958,E2 -1191.958} C_VEL
LIN {X 0,Y 594.391,Z 364.94,A -85,B 0,C 180,E1 -1194.446,E2 -1194.446} C_VEL
LIN {X 0,Y 594.388,Z 364.94,A -85,B 0,C 180,E1 -1196.699,E2 -1196.699} C_VEL
LIN {X 0,Y 594.383,Z 364.943,A -85,B 0,C 180,E1 -1198.998,E2 -1198.998} C_VEL
LIN {X 0,Y 594.393,Z 364.946,A -85,B 0,C 180,E1 -1201.645,E2 -1201.645} C_VEL
LIN {X 0,Y 594.4,Z 364.939,A -85,B 0,C 180,E1 -1204.578,E2 -1204.578} C_VEL
LIN {X 0,Y 594.387,Z 364.946,A -85,B 0,C 180,E1 -1207.086,E2 -1207.086} C_VEL
LIN {X 0,Y 594.377,Z 364.944,A -85,B 0,C 180,E1 -1209.774,E2 -1209.774} C_VEL
LIN {X 0,Y 594.367,Z 364.943,A -85,B 0,C 180,E1 -1212.375,E2 -1212.375} C_VEL
LIN {X 0,Y 594.362,Z 364.953,A -85,B 0,C 180,E1 -1215.191,E2 -1215.191} C_VEL
LIN {X 0,Y 594.386,Z 364.943,A -85,B 0,C 180,E1 -1217.626,E2 -1217.626} C_VEL
LIN {X 0,Y 594.39,Z 364.94,A -85,B 0,C 180,E1 -1220.32,E2 -1220.32} C_VEL
LIN {X 0,Y 594.386,Z 364.948,A -85,B 0,C 180,E1 -1222.913,E2 -1222.913} C_VEL
LIN {X 0,Y 594.381,Z 364.941,A -85,B 0,C 180,E1 -1225.86,E2 -1225.86} C_VEL
LIN {X 0,Y 594.386,Z 364.945,A -85,B 0,C 180,E1 -1228.651,E2 -1228.651} C_VEL
LIN {X 0,Y 594.38,Z 364.949,A -85,B 0,C 180,E1 -1231.041,E2 -1231.041} C_VEL
LIN {X 0,Y 594.384,Z 364.94,A -85,B 0,C 180,E1 -1233.976,E2 -1233.976} C_VEL
LIN {X 0,Y 594.384,Z 364.943,A -85,B 0,C 180,E1 -1236.296,E2 -1236.296} C_VEL
LIN {X 0,Y 594.401,Z 364.941,A -85,B 0,C 180,E1 -1239.224,E2 -1239.224} C_VEL
LIN {X 0,Y 594.377,Z 364.943,A -85,B 0,C 180,E1 -1242.096,E2 -1242.096} C_VEL
LIN {X 0,Y 594.365,Z 364.946,A -85,B 0,C 180,E1 -1244.219,E2 -1244.219} C_VEL
LIN {X 0,Y 594.365,Z 364.947,A -85,B 0,C 180,E1 -1247.017,E2 -1247.017} C_VEL
LIN {X 0,Y 594.389,Z 364.94,A -85,B 0,C 180,E1 -1249.784,E2 -1249.784} C_VEL
LIN {X 0,Y 594.396,Z 364.949,A -85,B 0,C 180,E1 -1252.527,E2 -1252.527} C_VEL
LIN {X 0,Y 594.395,Z 364.94,A -85,B 0,C 180,E1 -1255.252,E2 -1255.252} C_VEL
LIN {X 0,Y 594.389,Z 364.943,A -85,B 0,C 180,E1 -1257.967,E2 -1257.967} C_VEL
LIN {X 0,Y 594.419,Z 364.941,A -85,B 0,C 180,E1 -1260.677,E2 -1260.677} C_VEL
LIN {X 0,Y 594.38,Z 364.941,A -85,B 0,C 180,E1 -1263.389,E2 -1263.389} C_VEL
LIN {X 0,Y 594.365,Z 364.95,A -85,B 0,C 180,E1 -1266.109,E2 -1266.109} C_VEL
LIN {X 0,Y 594.395,Z 364.941,A -85,B 0,C 180,E1 -1268.842,E2 -1268.842} C_VEL
LIN {X 0,Y 594.388,Z 364.942,A -85,B 0,C 180,E1 -1271.596,E2 -1271.596} C_VEL
LIN {X 0,Y 594.384,Z 364.947,A -85,B 0,C 180,E1 -1274.377,E2 -1274.377} C_VEL
LIN {X 0,Y 594.365,Z 364.943,A -85,B 0,C 180,E1 -1275.337,E2 -1275.337} C_VEL
LIN {X 0,Y 593.7,Z 365.033,A -85,B 0,C 180,E1 -1275.903,E2 -1275.903} C_VEL
LIN {X 0,Y 590.846,Z 365.393,A -85,B 0,C 180,E1 -1276.821,E2 -1276.821} C_VEL
LIN {X 0,Y 588.436,Z 365.694,A -85,B 0,C 180,E1 -1277.56,E2 -1277.56} C_VEL
LIN {X 0,Y 587.405,Z 365.819,A -85,B 0,C 180,E1 -1278.13,E2 -1278.13} C_VEL
LIN {X 0,Y 587.323,Z 365.826,A -85,B 0,C 180,E1 -1278.323,E2 -1278.323} C_VEL
LIN {X 0,Y 587.352,Z 365.817,A -85,B 0,C 180,E1 -1281.045,E2 -1281.045} C_VEL
LIN {X 0,Y 587.337,Z 365.828,A -85,B 0,C 180,E1 -1284.006,E2 -1284.006} C_VEL
LIN {X 0,Y 587.359,Z 365.82,A -85,B 0,C 180,E1 -1286.278,E2 -1286.278} C_VEL
LIN {X 0,Y 587.348,Z 365.818,A -85,B 0,C 180,E1 -1289.135,E2 -1289.135} C_VEL
LIN {X 0,Y 587.355,Z 365.826,A -85,B 0,C 180,E1 -1291.839,E2 -1291.839} C_VEL
LIN {X 0,Y 587.352,Z 365.818,A -85,B 0,C 180,E1 -1294.35,E2 -1294.35} C_VEL
LIN {X 0,Y 587.349,Z 365.817,A -85,B 0,C 180,E1 -1296.747,E2 -1296.747} C_VEL
LIN {X 0,Y 587.344,Z 365.823,A -85,B 0,C 180,E1 -1299.36,E2 -1299.36} C_VEL
LIN {X 0,Y 587.331,Z 365.822,A -85,B 0,C 180,E1 -1302.108,E2 -1302.108} C_VEL
LIN {X 0,Y 587.313,Z 365.824,A -85,B 0,C 180,E1 -1305.089,E2 -1305.089} C_VEL
LIN {X 0,Y 587.35,Z 365.82,A -85,B 0,C 180,E1 -1307.928,E2 -1307.928} C_VEL
LIN {X 0,Y 587.333,Z 365.823,A -85,B 0,C 180,E1 -1311.058,E2 -1311.058} C_VEL
LIN {X 0,Y 587.353,Z 365.824,A -85,B 0,C 180,E1 -1313.292,E2 -1313.292} C_VEL
LIN {X 0,Y 587.368,Z 365.818,A -85,B 0,C 180,E1 -1315.781,E2 -1315.781} C_VEL
LIN {X 0,Y 587.347,Z 365.817,A -85,B 0,C 180,E1 -1318.232,E2 -1318.232} C_VEL
LIN {X 0,Y 587.351,Z 365.82,A -85,B 0,C 180,E1 -1320.867,E2 -1320.867} C_VEL
LIN {X 0,Y 587.36,Z 365.817,A -85,B 0,C 180,E1 -1323.819,E2 -1323.819} C_VEL
LIN {X 0,Y 587.336,Z 365.819,A -85,B 0,C 180,E1 -1325.994,E2 -1325.994} C_VEL
LIN {X 0,Y 587.319,Z 365.82,A -85,B 0,C 180,E1 -1328.226,E2 -1328.226} C_VEL
LIN {X 0,Y 587.349,Z 365.826,A -85,B 0,C 180,E1 -1331.151,E2 -1331.151} C_VEL
LIN {X 0,Y 587.323,Z 365.82,A -85,B 0,C 180,E1 -1334.025,E2 -1334.025} C_VEL
LIN {X 0,Y 587.362,Z 365.815,A -85,B 0,C 180,E1 -1336.154,E2 -1336.154} C_VEL
LIN {X 0,Y 587.343,Z 365.828,A -85,B 0,C 180,E1 -1338.963,E2 -1338.963} C_VEL
LIN {X 0,Y 587.367,Z 365.82,A -85,B 0,C 180,E1 -1341.745,E2 -1341.745} C_VEL
LIN {X 0,Y 587.387,Z 365.97,A -85,B 0,C 180,E1 -1342.567,E2 -1342.567} C_VEL
LIN {X 0,Y 587.588,Z 374.484,A -85,B 0,C 180,E1 -1343.993,E2 -1343.993} C_VEL
LIN {X 0,Y 587.457,Z 391.345,A -85,B 0,C 180,E1 -1346.742,E2 -1346.742} C_VEL
LIN {X 0,Y 587.385,Z 408.595,A -85,B 0,C 180,E1 -1349.507,E2 -1349.507} C_VEL
LIN {X 0,Y 587.566,Z 410.198,A -85,B 0,C 180,E1 -1349.582,E2 -1349.582} C_VEL
LIN {X 0,Y 587.857,Z 415.753,A -85,B 0,C 180,E1 -1349.657,E2 -1349.657} C_VEL
LIN {X 0,Y 587.734,Z 515.884,A -85,B 0,C 180,E1 -1350.899,E2 -1350.899} C_VEL
LIN {X 0,Y 587.714,Z 528.959,A -85,B 0,C 180,E1 -1351.199,E2 -1351.199} C_VEL
LIN {X 0,Y 587.579,Z 541.584,A -85,B 0,C 180,E1 -1351.628,E2 -1351.628} C_VEL
LIN {X 0,Y 587.525,Z 552.807,A -85,B 0,C 180,E1 -1352.142,E2 -1352.142} C_VEL
LIN {X 0,Y 587.453,Z 564.422,A -85,B 0,C 180,E1 -1352.828,E2 -1352.828} C_VEL
LIN {X 0,Y 587.38,Z 575.896,A -85,B 0,C 180,E1 -1353.687,E2 -1353.687} C_VEL
LIN {X 0,Y 587.332,Z 584.296,A -85,B 0,C 180,E1 -1354.461,E2 -1354.461} C_VEL
LIN {X 0,Y 587.238,Z 593.439,A -85,B 0,C 180,E1 -1355.494,E2 -1355.494} C_VEL
LIN {X 0,Y 587.22,Z 601.301,A -85,B 0,C 180,E1 -1356.603,E2 -1356.603} C_VEL
LIN {X 0,Y 587.197,Z 606.756,A -85,B 0,C 180,E1 -1357.565,E2 -1357.565} C_VEL
LIN {X 0,Y 587.19,Z 611.458,A -85,B 0,C 180,E1 -1358.604,E2 -1358.604} C_VEL
LIN {X 0,Y 587.159,Z 615.057,A -85,B 0,C 180,E1 -1359.646,E2 -1359.646} C_VEL
LIN {X 0,Y 587.143,Z 616.908,A -85,B 0,C 180,E1 -1360.343,E2 -1360.343} C_VEL
LIN {X 0,Y 587.164,Z 618.288,A -85,B 0,C 180,E1 -1361.041,E2 -1361.041} C_VEL
LIN {X 0,Y 587.154,Z 619.261,A -85,B 0,C 180,E1 -1361.74,E2 -1361.74} C_VEL
LIN {X 0,Y 587.159,Z 619.84,A -85,B 0,C 180,E1 -1362.442,E2 -1362.442} C_VEL
LIN {X 0,Y 587.145,Z 619.983,A -85,B 0,C 180,E1 -1363.145,E2 -1363.145} C_VEL
LIN {X 0,Y 587.158,Z 619.454,A -85,B 0,C 180,E1 -1364.18,E2 -1364.18} C_VEL
LIN {X 0,Y 587.131,Z 617.912,A -85,B 0,C 180,E1 -1365.268,E2 -1365.268} C_VEL
LIN {X 0,Y 587.151,Z 615.384,A -85,B 0,C 180,E1 -1366.337,E2 -1366.337} C_VEL
LIN {X 0,Y 587.17,Z 611.768,A -85,B 0,C 180,E1 -1367.411,E2 -1367.411} C_VEL
LIN {X 0,Y 587.209,Z 606.934,A -85,B 0,C 180,E1 -1368.491,E2 -1368.491} C_VEL
LIN {X 0,Y 587.239,Z 600.709,A -85,B 0,C 180,E1 -1369.578,E2 -1369.578} C_VEL
LIN {X 0,Y 587.283,Z 592.84,A -85,B 0,C 180,E1 -1370.672,E2 -1370.672} C_VEL
LIN {X 0,Y 587.313,Z 584.697,A -85,B 0,C 180,E1 -1371.59,E2 -1371.59} C_VEL
LIN {X 0,Y 587.415,Z 574.582,A -85,B 0,C 180,E1 -1372.51,E2 -1372.51} C_VEL
LIN {X 0,Y 587.447,Z 564.553,A -85,B 0,C 180,E1 -1373.253,E2 -1373.253} C_VEL
LIN {X 0,Y 587.533,Z 553.647,A -85,B 0,C 180,E1 -1373.904,E2 -1373.904} C_VEL
LIN {X 0,Y 587.623,Z 541.236,A -85,B 0,C 180,E1 -1374.475,E2 -1374.475} C_VEL
LIN {X 0,Y 587.682,Z 528.395,A -85,B 0,C 180,E1 -1374.908,E2 -1374.908} C_VEL
LIN {X 0,Y 587.736,Z 515.971,A -85,B 0,C 180,E1 -1375.189,E2 -1375.189} C_VEL
LIN {X 0,Y 587.719,Z 411.207,A -85,B 0,C 180,E1 -1376.492,E2 -1376.492} C_VEL
LIN {X 0,Y 587.369,Z 408.891,A -85,B 0,C 180,E1 -1376.556,E2 -1376.556} C_VEL
LIN {X 0,Y 587.435,Z 392.581,A -85,B 0,C 180,E1 -1379.148,E2 -1379.148} C_VEL
LIN {X 0,Y 587.571,Z 375.865,A -85,B 0,C 180,E1 -1381.871,E2 -1381.871} C_VEL
LIN {X 0,Y 587.525,Z 366.716,A -85,B 0,C 180,E1 -1383.383,E2 -1383.383} C_VEL
LIN {X 0,Y 587.338,Z 365.847,A -85,B 0,C 180,E1 -1383.601,E2 -1383.601} C_VEL
LIN {X 0,Y 587.355,Z 365.818,A -85,B 0,C 180,E1 -1385.894,E2 -1385.894} C_VEL
LIN {X 0,Y 587.332,Z 365.82,A -85,B 0,C 180,E1 -1388.478,E2 -1388.478} C_VEL
LIN {X 0,Y 587.335,Z 365.828,A -85,B 0,C 180,E1 -1391.156,E2 -1391.156} C_VEL
LIN {X 0,Y 587.329,Z 365.819,A -85,B 0,C 180,E1 -1394.113,E2 -1394.113} C_VEL
LIN {X 0,Y 587.333,Z 365.827,A -85,B 0,C 180,E1 -1396.995,E2 -1396.995} C_VEL
LIN {X 0,Y 587.324,Z 365.821,A -85,B 0,C 180,E1 -1399.746,E2 -1399.746} C_VEL
LIN {X 0,Y 587.342,Z 365.818,A -85,B 0,C 180,E1 -1402.392,E2 -1402.392} C_VEL
LIN {X 0,Y 587.345,Z 365.825,A -85,B 0,C 180,E1 -1404.946,E2 -1404.946} C_VEL
LIN {X 0,Y 587.336,Z 365.822,A -85,B 0,C 180,E1 -1407.421,E2 -1407.421} C_VEL
LIN {X 0,Y 587.339,Z 365.816,A -85,B 0,C 180,E1 -1409.83,E2 -1409.83} C_VEL
LIN {X 0,Y 587.343,Z 365.818,A -85,B 0,C 180,E1 -1412.306,E2 -1412.306} C_VEL
LIN {X 0,Y 587.333,Z 365.821,A -85,B 0,C 180,E1 -1414.483,E2 -1414.483} C_VEL
LIN {X 0,Y 587.361,Z 365.817,A -85,B 0,C 180,E1 -1417.487,E2 -1417.487} C_VEL
LIN {X 0,Y 587.339,Z 365.82,A -85,B 0,C 180,E1 -1420.425,E2 -1420.425} C_VEL
LIN {X 0,Y 587.349,Z 365.821,A -85,B 0,C 180,E1 -1423.311,E2 -1423.311} C_VEL
LIN {X 0,Y 587.354,Z 365.816,A -85,B 0,C 180,E1 -1426.154,E2 -1426.154} C_VEL
LIN {X 0,Y 587.342,Z 365.826,A -85,B 0,C 180,E1 -1428.962,E2 -1428.962} C_VEL
LIN {X 0,Y 587.364,Z 365.815,A -85,B 0,C 180,E1 -1431.745,E2 -1431.745} C_VEL
LIN {X 0,Y 587.358,Z 365.819,A -85,B 0,C 180,E1 -1434.507,E2 -1434.507} C_VEL
LIN {X 0,Y 587.377,Z 365.816,A -85,B 0,C 180,E1 -1437.257,E2 -1437.257} C_VEL
LIN {X 0,Y 587.373,Z 365.813,A -85,B 0,C 180,E1 -1440,E2 -1440} C_VEL
LIN {X 0,Y 587.378,Z 365.822,A -85,B 0,C 180,E1 -1442.743,E2 -1442.743} C_VEL
LIN {X 0,Y 587.356,Z 365.816,A -85,B 0,C 180,E1 -1445.493,E2 -1445.493} C_VEL
LIN {X 0,Y 587.365,Z 365.816,A -85,B 0,C 180,E1 -1448.255,E2 -1448.255} C_VEL
LIN {X 0,Y 587.352,Z 365.82,A -85,B 0,C 180,E1 -1451.142,E2 -1451.142} C_VEL
LIN {X 0,Y 587.355,Z 365.818,A -85,B 0,C 180,E1 -1454.261,E2 -1454.261} C_VEL
LIN {X 0,Y 587.354,Z 365.816,A -85,B 0,C 180,E1 -1457.406,E2 -1457.406} C_VEL
LIN {X 0,Y 587.33,Z 365.822,A -85,B 0,C 180,E1 -1460.305,E2 -1460.305} C_VEL
LIN {X 0,Y 587.359,Z 365.817,A -85,B 0,C 180,E1 -1463.257,E2 -1463.257} C_VEL
LIN {X 0,Y 587.356,Z 365.819,A -85,B 0,C 180,E1 -1466.278,E2 -1466.278} C_VEL
LIN {X 0,Y 587.347,Z 365.819,A -85,B 0,C 180,E1 -1469.135,E2 -1469.135} C_VEL
LIN {X 0,Y 587.352,Z 365.816,A -85,B 0,C 180,E1 -1471.839,E2 -1471.839} C_VEL
LIN {X 0,Y 587.352,Z 365.822,A -85,B 0,C 180,E1 -1474.35,E2 -1474.35} C_VEL
LIN {X 0,Y 587.348,Z 365.824,A -85,B 0,C 180,E1 -1476.747,E2 -1476.747} C_VEL
LIN {X 0,Y 587.341,Z 365.818,A -85,B 0,C 180,E1 -1479.36,E2 -1479.36} C_VEL
LIN {X 0,Y 587.333,Z 365.82,A -85,B 0,C 180,E1 -1482.109,E2 -1482.109} C_VEL
LIN {X 0,Y 587.311,Z 365.823,A -85,B 0,C 180,E1 -1485.09,E2 -1485.09} C_VEL
LIN {X 0,Y 587.349,Z 365.818,A -85,B 0,C 180,E1 -1487.928,E2 -1487.928} C_VEL
LIN {X 0,Y 587.333,Z 365.821,A -85,B 0,C 180,E1 -1491.059,E2 -1491.059} C_VEL
LIN {X 0,Y 587.352,Z 365.816,A -85,B 0,C 180,E1 -1493.292,E2 -1493.292} C_VEL
LIN {X 0,Y 587.369,Z 365.815,A -85,B 0,C 180,E1 -1495.781,E2 -1495.781} C_VEL
LIN {X 0,Y 587.352,Z 365.823,A -85,B 0,C 180,E1 -1498.233,E2 -1498.233} C_VEL
LIN {X 0,Y 587.35,Z 365.82,A -85,B 0,C 180,E1 -1500.867,E2 -1500.867} C_VEL
LIN {X 0,Y 587.362,Z 365.817,A -85,B 0,C 180,E1 -1503.819,E2 -1503.819} C_VEL
LIN {X 0,Y 587.338,Z 365.823,A -85,B 0,C 180,E1 -1505.994,E2 -1505.994} C_VEL
LIN {X 0,Y 587.369,Z 366.03,A -85,B 0,C 180,E1 -1507.951,E2 -1507.951} C_VEL
LIN {X 0,Y 587.749,Z 370.357,A -85,B 0,C 180,E1 -1508.645,E2 -1508.645} C_VEL
LIN {X 0,Y 587.579,Z 388.234,A -85,B 0,C 180,E1 -1511.34,E2 -1511.34} C_VEL
LIN {X 0,Y 587.491,Z 405.127,A -85,B 0,C 180,E1 -1513.852,E2 -1513.852} C_VEL
LIN {X 0,Y 587.409,Z 423.28,A -85,B 0,C 180,E1 -1516.487,E2 -1516.487} C_VEL
LIN {X 0,Y 587.871,Z 426.756,A -85,B 0,C 180,E1 -1516.564,E2 -1516.564} C_VEL
LIN {X 0,Y 587.754,Z 530.969,A -85,B 0,C 180,E1 -1517.856,E2 -1517.856} C_VEL
LIN {X 0,Y 587.685,Z 544.233,A -85,B 0,C 180,E1 -1518.161,E2 -1518.161} C_VEL
LIN {X 0,Y 587.64,Z 556.771,A -85,B 0,C 180,E1 -1518.591,E2 -1518.591} C_VEL
LIN {X 0,Y 587.554,Z 568.638,A -85,B 0,C 180,E1 -1519.141,E2 -1519.141} C_VEL
LIN {X 0,Y 587.465,Z 580.207,A -85,B 0,C 180,E1 -1519.837,E2 -1519.837} C_VEL
LIN {X 0,Y 587.391,Z 590.602,A -85,B 0,C 180,E1 -1520.618,E2 -1520.618} C_VEL
LIN {X 0,Y 587.321,Z 599.116,A -85,B 0,C 180,E1 -1521.398,E2 -1521.398} C_VEL
LIN {X 0,Y 587.273,Z 606.963,A -85,B 0,C 180,E1 -1522.263,E2 -1522.263} C_VEL
LIN {X 0,Y 587.23,Z 613.472,A -85,B 0,C 180,E1 -1523.127,E2 -1523.127} C_VEL
LIN {X 0,Y 587.236,Z 619.868,A -85,B 0,C 180,E1 -1524.162,E2 -1524.162} C_VEL
LIN {X 0,Y 587.147,Z 624.951,A -85,B 0,C 180,E1 -1525.194,E2 -1525.194} C_VEL
LIN {X 0,Y 587.212,Z 628.896,A -85,B 0,C 180,E1 -1526.226,E2 -1526.226} C_VEL
LIN {X 0,Y 587.132,Z 631.809,A -85,B 0,C 180,E1 -1527.256,E2 -1527.256} C_VEL
LIN {X 0,Y 587.139,Z 633.201,A -85,B 0,C 180,E1 -1527.942,E2 -1527.942} C_VEL
LIN {X 0,Y 587.14,Z 634.784,A -85,B 0,C 180,E1 -1529.314,E2 -1529.314} C_VEL
LIN {X 0,Y 587.137,Z 635,A -85,B 0,C 180,E1 -1530,E2 -1530} C_VEL
LIN {X 0,Y 587.147,Z 634.185,A -85,B 0,C 180,E1 -1531.372,E2 -1531.372} C_VEL
LIN {X 0,Y 587.139,Z 633.201,A -85,B 0,C 180,E1 -1532.058,E2 -1532.058} C_VEL
LIN {X 0,Y 587.132,Z 631.809,A -85,B 0,C 180,E1 -1532.744,E2 -1532.744} C_VEL
LIN {X 0,Y 587.212,Z 628.896,A -85,B 0,C 180,E1 -1533.774,E2 -1533.774} C_VEL
LIN {X 0,Y 587.147,Z 624.949,A -85,B 0,C 180,E1 -1534.806,E2 -1534.806} C_VEL
LIN {X 0,Y 587.217,Z 618.877,A -85,B 0,C 180,E1 -1536.011,E2 -1536.011} C_VEL
LIN {X 0,Y 587.245,Z 612.236,A -85,B 0,C 180,E1 -1537.046,E2 -1537.046} C_VEL
LIN {X 0,Y 587.299,Z 603.99,A -85,B 0,C 180,E1 -1538.083,E2 -1538.083} C_VEL
LIN {X 0,Y 587.343,Z 595.538,A -85,B 0,C 180,E1 -1538.949,E2 -1538.949} C_VEL
LIN {X 0,Y 587.416,Z 585.096,A -85,B 0,C 180,E1 -1539.816,E2 -1539.816} C_VEL
LIN {X 0,Y 587.49,Z 574.758,A -85,B 0,C 180,E1 -1540.511,E2 -1540.511} C_VEL
LIN {X 0,Y 587.584,Z 562.802,A -85,B 0,C 180,E1 -1541.149,E2 -1541.149} C_VEL
LIN {X 0,Y 587.637,Z 550.592,A -85,B 0,C 180,E1 -1541.639,E2 -1541.639} C_VEL
LIN {X 0,Y 587.701,Z 537.439,A -85,B 0,C 180,E1 -1542.014,E2 -1542.014} C_VEL
LIN {X 0,Y 587.775,Z 525.09,A -85,B 0,C 180,E1 -1542.231,E2 -1542.231} C_VEL
LIN {X 0,Y 587.687,Z 425.161,A -85,B 0,C 180,E1 -1543.46,E2 -1543.46} C_VEL
LIN {X 0,Y 587.41,Z 423.272,A -85,B 0,C 180,E1 -1543.514,E2 -1543.514} C_VEL
LIN {X 0,Y 587.504,Z 403.918,A -85,B 0,C 180,E1 -1546.327,E2 -1546.327} C_VEL
LIN {X 0,Y 587.606,Z 387.025,A -85,B 0,C 180,E1 -1548.84,E2 -1548.84} C_VEL
LIN {X 0,Y 587.766,Z 368.921,A -85,B 0,C 180,E1 -1551.573,E2 -1551.573} C_VEL
LIN {X 0,Y 587.354,Z 365.876,A -85,B 0,C 180,E1 -1552.096,E2 -1552.096} C_VEL
LIN {X 0,Y 587.355,Z 365.818,A -85,B 0,C 180,E1 -1554.758,E2 -1554.758} C_VEL
LIN {X 0,Y 587.332,Z 365.822,A -85,B 0,C 180,E1 -1557.046,E2 -1557.046} C_VEL
LIN {X 0,Y 587.35,Z 365.826,A -85,B 0,C 180,E1 -1559.379,E2 -1559.379} C_VEL
LIN {X 0,Y 587.355,Z 365.819,A -85,B 0,C 180,E1 -1561.837,E2 -1561.837} C_VEL
LIN {X 0,Y 587.358,Z 365.815,A -85,B 0,C 180,E1 -1564.349,E2 -1564.349} C_VEL
LIN {X 0,Y 587.353,Z 365.818,A -85,B 0,C 180,E1 -1566.746,E2 -1566.746} C_VEL
LIN {X 0,Y 587.347,Z 365.826,A -85,B 0,C 180,E1 -1569.358,E2 -1569.358} C_VEL
LIN {X 0,Y 587.333,Z 365.819,A -85,B 0,C 180,E1 -1572.107,E2 -1572.107} C_VEL
LIN {X 0,Y 587.314,Z 365.83,A -85,B 0,C 180,E1 -1575.088,E2 -1575.088} C_VEL
LIN {X 0,Y 587.35,Z 365.817,A -85,B 0,C 180,E1 -1577.927,E2 -1577.927} C_VEL
LIN {X 0,Y 587.344,Z 365.821,A -85,B 0,C 180,E1 -1580.64,E2 -1580.64} C_VEL
LIN {X 0,Y 587.351,Z 365.823,A -85,B 0,C 180,E1 -1583.291,E2 -1583.291} C_VEL
LIN {X 0,Y 587.364,Z 365.815,A -85,B 0,C 180,E1 -1585.78,E2 -1585.78} C_VEL
LIN {X 0,Y 587.35,Z 365.817,A -85,B 0,C 180,E1 -1588.231,E2 -1588.231} C_VEL
LIN {X 0,Y 587.345,Z 365.827,A -85,B 0,C 180,E1 -1590.866,E2 -1590.866} C_VEL
LIN {X 0,Y 587.356,Z 365.816,A -85,B 0,C 180,E1 -1593.818,E2 -1593.818} C_VEL
LIN {X 0,Y 587.331,Z 365.819,A -85,B 0,C 180,E1 -1595.993,E2 -1595.993} C_VEL
LIN {X 0,Y 587.342,Z 365.825,A -85,B 0,C 180,E1 -1598.963,E2 -1598.963} C_VEL
LIN {X 0,Y 587.324,Z 365.82,A -85,B 0,C 180,E1 -1601.873,E2 -1601.873} C_VEL
LIN {X 0,Y 587.323,Z 365.822,A -85,B 0,C 180,E1 -1604.025,E2 -1604.025} C_VEL
LIN {X 0,Y 587.354,Z 365.819,A -85,B 0,C 180,E1 -1606.154,E2 -1606.154} C_VEL
LIN {X 0,Y 587.338,Z 365.822,A -85,B 0,C 180,E1 -1608.962,E2 -1608.962} C_VEL
LIN {X 0,Y 587.364,Z 365.816,A -85,B 0,C 180,E1 -1611.745,E2 -1611.745} C_VEL
LIN {X 0,Y 587.353,Z 365.826,A -85,B 0,C 180,E1 -1614.507,E2 -1614.507} C_VEL
LIN {X 0,Y 587.374,Z 365.814,A -85,B 0,C 180,E1 -1617.257,E2 -1617.257} C_VEL
LIN {X 0,Y 587.376,Z 365.818,A -85,B 0,C 180,E1 -1620,E2 -1620} C_VEL
LIN {X 0,Y 587.374,Z 365.818,A -85,B 0,C 180,E1 -1622.743,E2 -1622.743} C_VEL
LIN {X 0,Y 587.354,Z 365.817,A -85,B 0,C 180,E1 -1625.493,E2 -1625.493} C_VEL
LIN {X 0,Y 587.365,Z 365.824,A -85,B 0,C 180,E1 -1628.255,E2 -1628.255} C_VEL
LIN {X 0,Y 587.34,Z 365.818,A -85,B 0,C 180,E1 -1631.134,E2 -1631.134} C_VEL
LIN {X 0,Y 587.355,Z 365.822,A -85,B 0,C 180,E1 -1633.846,E2 -1633.846} C_VEL
LIN {X 0,Y 587.359,Z 365.816,A -85,B 0,C 180,E1 -1636.82,E2 -1636.82} C_VEL
LIN {X 0,Y 587.323,Z 365.826,A -85,B 0,C 180,E1 -1638.323,E2 -1638.323} C_VEL
LIN {X 0,Y 586.668,Z 365.904,A -85,B 0,C 180,E1 -1638.895,E2 -1638.895} C_VEL
LIN {X 0,Y 583.836,Z 366.261,A -85,B 0,C 180,E1 -1639.823,E2 -1639.823} C_VEL
LIN {X 0,Y 581.428,Z 366.558,A -85,B 0,C 180,E1 -1640.57,E2 -1640.57} C_VEL
LIN {X 0,Y 580.377,Z 366.687,A -85,B 0,C 180,E1 -1641.146,E2 -1641.146} C_VEL
LIN {X 0,Y 580.283,Z 366.698,A -85,B 0,C 180,E1 -1641.342,E2 -1641.342} C_VEL
LIN {X 0,Y 580.297,Z 366.7,A -85,B 0,C 180,E1 -1644.316,E2 -1644.316} C_VEL
LIN {X 0,Y 580.302,Z 366.696,A -85,B 0,C 180,E1 -1646.622,E2 -1646.622} C_VEL
LIN {X 0,Y 580.303,Z 366.697,A -85,B 0,C 180,E1 -1649.312,E2 -1649.312} C_VEL
LIN {X 0,Y 580.301,Z 366.699,A -85,B 0,C 180,E1 -1652.2,E2 -1652.2} C_VEL
LIN {X 0,Y 580.296,Z 366.696,A -85,B 0,C 180,E1 -1654.696,E2 -1654.696} C_VEL
LIN {X 0,Y 580.297,Z 366.699,A -85,B 0,C 180,E1 -1657.269,E2 -1657.269} C_VEL
LIN {X 0,Y 580.296,Z 366.697,A -85,B 0,C 180,E1 -1660.272,E2 -1660.272} C_VEL
LIN {X 0,Y 580.279,Z 366.698,A -85,B 0,C 180,E1 -1662.706,E2 -1662.706} C_VEL
LIN {X 0,Y 580.267,Z 366.708,A -85,B 0,C 180,E1 -1665.61,E2 -1665.61} C_VEL
LIN {X 0,Y 580.312,Z 366.694,A -85,B 0,C 180,E1 -1668.235,E2 -1668.235} C_VEL
LIN {X 0,Y 580.289,Z 366.699,A -85,B 0,C 180,E1 -1670.967,E2 -1670.967} C_VEL
LIN {X 0,Y 580.296,Z 366.703,A -85,B 0,C 180,E1 -1673.599,E2 -1673.599} C_VEL
LIN {X 0,Y 580.32,Z 366.693,A -85,B 0,C 180,E1 -1676.146,E2 -1676.146} C_VEL
LIN {X 0,Y 580.282,Z 366.698,A -85,B 0,C 180,E1 -1678.615,E2 -1678.615} C_VEL
LIN {X 0,Y 580.294,Z 366.701,A -85,B 0,C 180,E1 -1681.024,E2 -1681.024} C_VEL
LIN {X 0,Y 580.292,Z 366.699,A -85,B 0,C 180,E1 -1683.666,E2 -1683.666} C_VEL
LIN {X 0,Y 580.301,Z 366.697,A -85,B 0,C 180,E1 -1685.684,E2 -1685.684} C_VEL
LIN {X 0,Y 580.27,Z 366.699,A -85,B 0,C 180,E1 -1687.948,E2 -1687.948} C_VEL
LIN {X 0,Y 580.298,Z 366.702,A -85,B 0,C 180,E1 -1690.914,E2 -1690.914} C_VEL
LIN {X 0,Y 580.277,Z 366.698,A -85,B 0,C 180,E1 -1693.826,E2 -1693.826} C_VEL
LIN {X 0,Y 580.328,Z 366.691,A -85,B 0,C 180,E1 -1695.983,E2 -1695.983} C_VEL
LIN {X 0,Y 580.307,Z 366.703,A -85,B 0,C 180,E1 -1698.827,E2 -1698.827} C_VEL
LIN {X 0,Y 580.33,Z 366.697,A -85,B 0,C 180,E1 -1701.644,E2 -1701.644} C_VEL
LIN {X 0,Y 580.375,Z 366.939,A -85,B 0,C 180,E1 -1702.477,E2 -1702.477} C_VEL
LIN {X 0,Y 580.611,Z 375.477,A -85,B 0,C 180,E1 -1703.92,E2 -1703.92} C_VEL
LIN {X 0,Y 580.448,Z 392.338,A -85,B 0,C 180,E1 -1706.703,E2 -1706.703} C_VEL
LIN {X 0,Y 580.367,Z 408.682,A -85,B 0,C 180,E1 -1709.349,E2 -1709.349} C_VEL
LIN {X 0,Y 580.517,Z 410.114,A -85,B 0,C 180,E1 -1709.415,E2 -1709.415} C_VEL
LIN {X 0,Y 580.975,Z 414.488,A -85,B 0,C 180,E1 -1709.48,E2 -1709.48} C_VEL
LIN {X 0,Y 580.806,Z 516.203,A -85,B 0,C 180,E1 -1710.758,E2 -1710.758} C_VEL
LIN {X 0,Y 580.747,Z 529.938,A -85,B 0,C 180,E1 -1711.083,E2 -1711.083} C_VEL
LIN {X 0,Y 580.602,Z 542.309,A -85,B 0,C 180,E1 -1711.517,E2 -1711.517} C_VEL
LIN {X 0,Y 580.552,Z 554.126,A -85,B 0,C 180,E1 -1712.081,E2 -1712.081} C_VEL
LIN {X 0,Y 580.45,Z 565.47,A -85,B 0,C 180,E1 -1712.776,E2 -1712.776} C_VEL
LIN {X 0,Y 580.381,Z 575.712,A -85,B 0,C 180,E1 -1713.558,E2 -1713.558} C_VEL
LIN {X 0,Y 580.274,Z 584.15,A -85,B 0,C 180,E1 -1714.341,E2 -1714.341} C_VEL
LIN {X 0,Y 580.175,Z 593.325,A -85,B 0,C 180,E1 -1715.387,E2 -1715.387} C_VEL
LIN {X 0,Y 580.131,Z 600.381,A -85,B 0,C 180,E1 -1716.38,E2 -1716.38} C_VEL
LIN {X 0,Y 580.124,Z 605.768,A -85,B 0,C 180,E1 -1717.308,E2 -1717.308} C_VEL
LIN {X 0,Y 580.11,Z 610.68,A -85,B 0,C 180,E1 -1718.359,E2 -1718.359} C_VEL
LIN {X 0,Y 580.08,Z 614.475,A -85,B 0,C 180,E1 -1719.413,E2 -1719.413} C_VEL
LIN {X 0,Y 580.061,Z 617.244,A -85,B 0,C 180,E1 -1720.471,E2 -1720.471} C_VEL
LIN {X 0,Y 580.073,Z 618.544,A -85,B 0,C 180,E1 -1721.177,E2 -1721.177} C_VEL
LIN {X 0,Y 580.053,Z 619.443,A -85,B 0,C 180,E1 -1721.886,E2 -1721.886} C_VEL
LIN {X 0,Y 580.049,Z 619.905,A -85,B 0,C 180,E1 -1722.597,E2 -1722.597} C_VEL
LIN {X 0,Y 580.059,Z 619.947,A -85,B 0,C 180,E1 -1723.309,E2 -1723.309} C_VEL
LIN {X 0,Y 580.049,Z 619.409,A -85,B 0,C 180,E1 -1724.234,E2 -1724.234} C_VEL
LIN {X 0,Y 580.03,Z 617.573,A -85,B 0,C 180,E1 -1725.459,E2 -1725.459} C_VEL
LIN {X 0,Y 580.066,Z 615.901,A -85,B 0,C 180,E1 -1726.18,E2 -1726.18} C_VEL
LIN {X 0,Y 580.07,Z 612.487,A -85,B 0,C 180,E1 -1727.267,E2 -1727.267} C_VEL
LIN {X 0,Y 580.1,Z 607.895,A -85,B 0,C 180,E1 -1728.36,E2 -1728.36} C_VEL
LIN {X 0,Y 580.15,Z 602.186,A -85,B 0,C 180,E1 -1729.422,E2 -1729.422} C_VEL
LIN {X 0,Y 580.18,Z 595.801,A -85,B 0,C 180,E1 -1730.38,E2 -1730.38} C_VEL
LIN {X 0,Y 580.285,Z 588.31,A -85,B 0,C 180,E1 -1731.305,E2 -1731.305} C_VEL
LIN {X 0,Y 580.316,Z 579.059,A -85,B 0,C 180,E1 -1732.237,E2 -1732.237} C_VEL
LIN {X 0,Y 580.404,Z 569.39,A -85,B 0,C 180,E1 -1733.034,E2 -1733.034} C_VEL
LIN {X 0,Y 580.486,Z 558.9,A -85,B 0,C 180,E1 -1733.738,E2 -1733.738} C_VEL
LIN {X 0,Y 580.611,Z 546.854,A -85,B 0,C 180,E1 -1734.372,E2 -1734.372} C_VEL
LIN {X 0,Y 580.715,Z 533.798,A -85,B 0,C 180,E1 -1734.886,E2 -1734.886} C_VEL
LIN {X 0,Y 580.767,Z 520.499,A -85,B 0,C 180,E1 -1735.249,E2 -1735.249} C_VEL
LIN {X 0,Y 580.826,Z 505.171,A -85,B 0,C 180,E1 -1735.486,E2 -1735.486} C_VEL
LIN {X 0,Y 580.869,Z 412.347,A -85,B 0,C 180,E1 -1736.639,E2 -1736.639} C_VEL
LIN {X 0,Y 580.365,Z 408.993,A -85,B 0,C 180,E1 -1736.715,E2 -1736.715} C_VEL
LIN {X 0,Y 580.454,Z 392.648,A -85,B 0,C 180,E1 -1739.336,E2 -1739.336} C_VEL
LIN {X 0,Y 580.617,Z 374.186,A -85,B 0,C 180,E1 -1742.385,E2 -1742.385} C_VEL
LIN {X 0,Y 580.579,Z 368.383,A -85,B 0,C 180,E1 -1743.357,E2 -1743.357} C_VEL
LIN {X 0,Y 580.32,Z 366.748,A -85,B 0,C 180,E1 -1743.679,E2 -1743.679} C_VEL
LIN {X 0,Y 580.294,Z 366.697,A -85,B 0,C 180,E1 -1746.401,E2 -1746.401} C_VEL
LIN {X 0,Y 580.308,Z 366.703,A -85,B 0,C 180,E1 -1749.187,E2 -1749.187} C_VEL
LIN {X 0,Y 580.31,Z 366.695,A -85,B 0,C 180,E1 -1751.765,E2 -1751.765} C_VEL
LIN {X 0,Y 580.264,Z 366.702,A -85,B 0,C 180,E1 -1754.625,E2 -1754.625} C_VEL
LIN {X 0,Y 580.306,Z 366.695,A -85,B 0,C 180,E1 -1757.625,E2 -1757.625} C_VEL
LIN {X 0,Y 580.294,Z 366.695,A -85,B 0,C 180,E1 -1760.067,E2 -1760.067} C_VEL
LIN {X 0,Y 580.297,Z 366.705,A -85,B 0,C 180,E1 -1763.064,E2 -1763.064} C_VEL
LIN {X 0,Y 580.299,Z 366.698,A -85,B 0,C 180,E1 -1765.44,E2 -1765.44} C_VEL
LIN {X 0,Y 580.304,Z 366.694,A -85,B 0,C 180,E1 -1767.967,E2 -1767.967} C_VEL
LIN {X 0,Y 580.301,Z 366.697,A -85,B 0,C 180,E1 -1770.688,E2 -1770.688} C_VEL
LIN {X 0,Y 580.321,Z 366.693,A -85,B 0,C 180,E1 -1773.657,E2 -1773.657} C_VEL
LIN {X 0,Y 580.294,Z 366.698,A -85,B 0,C 180,E1 -1776.443,E2 -1776.443} C_VEL
LIN {X 0,Y 580.277,Z 366.7,A -85,B 0,C 180,E1 -1779.437,E2 -1779.437} C_VEL
LIN {X 0,Y 580.277,Z 366.698,A -85,B 0,C 180,E1 -1781.645,E2 -1781.645} C_VEL
LIN {X 0,Y 580.278,Z 366.697,A -85,B 0,C 180,E1 -1783.826,E2 -1783.826} C_VEL
LIN {X 0,Y 580.276,Z 366.703,A -85,B 0,C 180,E1 -1786.696,E2 -1786.696} C_VEL
LIN {X 0,Y 580.299,Z 366.695,A -85,B 0,C 180,E1 -1789.533,E2 -1789.533} C_VEL
LIN {X 0,Y 580.333,Z 366.693,A -85,B 0,C 180,E1 -1792.345,E2 -1792.345} C_VEL
LIN {X 0,Y 580.336,Z 366.696,A -85,B 0,C 180,E1 -1795.137,E2 -1795.137} C_VEL
LIN {X 0,Y 580.33,Z 366.69,A -85,B 0,C 180,E1 -1797.918,E2 -1797.918} C_VEL
LIN {X 0,Y 580.365,Z 366.694,A -85,B 0,C 180,E1 -1800.694,E2 -1800.694} C_VEL
LIN {X 0,Y 580.286,Z 366.696,A -85,B 0,C 180,E1 -1803.472,E2 -1803.472} C_VEL
LIN {X 0,Y 580.321,Z 366.692,A -85,B 0,C 180,E1 -1805.56,E2 -1805.56} C_VEL
LIN {X 0,Y 580.328,Z 366.694,A -85,B 0,C 180,E1 -1808.356,E2 -1808.356} C_VEL
LIN {X 0,Y 580.323,Z 366.695,A -85,B 0,C 180,E1 -1811.209,E2 -1811.209} C_VEL
LIN {X 0,Y 580.318,Z 366.692,A -85,B 0,C 180,E1 -1814.017,E2 -1814.017} C_VEL
LIN {X 0,Y 580.309,Z 366.7,A -85,B 0,C 180,E1 -1816.917,E2 -1816.917} C_VEL
LIN {X 0,Y 580.302,Z 366.694,A -85,B 0,C 180,E1 -1819.823,E2 -1819.823} C_VEL
LIN {X 0,Y 580.322,Z 366.7,A -85,B 0,C 180,E1 -1822.801,E2 -1822.801} C_VEL
LIN {X 0,Y 580.301,Z 366.698,A -85,B 0,C 180,E1 -1825.08,E2 -1825.08} C_VEL
LIN {X 0,Y 580.313,Z 366.693,A -85,B 0,C 180,E1 -1827.864,E2 -1827.864} C_VEL
LIN {X 0,Y 580.287,Z 366.705,A -85,B 0,C 180,E1 -1830.697,E2 -1830.697} C_VEL
LIN {X 0,Y 580.299,Z 366.695,A -85,B 0,C 180,E1 -1833.318,E2 -1833.318} C_VEL
LIN {X 0,Y 580.32,Z 366.692,A -85,B 0,C 180,E1 -1835.768,E2 -1835.768} C_VEL
LIN {X 0,Y 580.284,Z 366.699,A -85,B 0,C 180,E1 -1838.147,E2 -1838.147} C_VEL
LIN {X 0,Y 580.315,Z 366.696,A -85,B 0,C 180,E1 -1840.842,E2 -1840.842} C_VEL
LIN {X 0,Y 580.286,Z 366.696,A -85,B 0,C 180,E1 -1843.657,E2 -1843.657} C_VEL
LIN {X 0,Y 580.281,Z 366.706,A -85,B 0,C 180,E1 -1846.609,E2 -1846.609} C_VEL
LIN {X 0,Y 580.298,Z 366.696,A -85,B 0,C 180,E1 -1849.158,E2 -1849.158} C_VEL
LIN {X 0,Y 580.288,Z 366.698,A -85,B 0,C 180,E1 -1851.928,E2 -1851.928} C_VEL
LIN {X 0,Y 580.308,Z 366.703,A -85,B 0,C 180,E1 -1854.458,E2 -1854.458} C_VEL
LIN {X 0,Y 580.291,Z 366.699,A -85,B 0,C 180,E1 -1856.976,E2 -1856.976} C_VEL
LIN {X 0,Y 580.302,Z 366.695,A -85,B 0,C 180,E1 -1859.426,E2 -1859.426} C_VEL
LIN {X 0,Y 580.299,Z 366.701,A -85,B 0,C 180,E1 -1862.142,E2 -1862.142} C_VEL
LIN {X 0,Y 580.31,Z 366.698,A -85,B 0,C 180,E1 -1864.921,E2 -1864.921} C_VEL
LIN {X 0,Y 580.313,Z 366.788,A -85,B 0,C 180,E1 -1867.762,E2 -1867.762} C_VEL
LIN {X 0,Y 580.82,Z 370.138,A -85,B 0,C 180,E1 -1868.344,E2 -1868.344} C_VEL
LIN {X 0,Y 580.651,Z 387.028,A -85,B 0,C 180,E1 -1870.926,E2 -1870.926} C_VEL
LIN {X 0,Y 580.51,Z 405.127,A -85,B 0,C 180,E1 -1873.652,E2 -1873.652} C_VEL
LIN {X 0,Y 580.388,Z 423.28,A -85,B 0,C 180,E1 -1876.32,E2 -1876.32} C_VEL
LIN {X 0,Y 580.976,Z 428.545,A -85,B 0,C 180,E1 -1876.423,E2 -1876.423} C_VEL
LIN {X 0,Y 580.815,Z 530.969,A -85,B 0,C 180,E1 -1877.709,E2 -1877.709} C_VEL
LIN {X 0,Y 580.756,Z 544.234,A -85,B 0,C 180,E1 -1878.018,E2 -1878.018} C_VEL
LIN {X 0,Y 580.669,Z 556.383,A -85,B 0,C 180,E1 -1878.437,E2 -1878.437} C_VEL
LIN {X 0,Y 580.564,Z 568.637,A -85,B 0,C 180,E1 -1879.009,E2 -1879.009} C_VEL
LIN {X 0,Y 580.442,Z 580.209,A -85,B 0,C 180,E1 -1879.713,E2 -1879.713} C_VEL
LIN {X 0,Y 580.341,Z 590.604,A -85,B 0,C 180,E1 -1880.503,E2 -1880.503} C_VEL
LIN {X 0,Y 580.271,Z 599.116,A -85,B 0,C 180,E1 -1881.293,E2 -1881.293} C_VEL
LIN {X 0,Y 580.221,Z 606.963,A -85,B 0,C 180,E1 -1882.168,E2 -1882.168} C_VEL
LIN {X 0,Y 580.153,Z 614.652,A -85,B 0,C 180,E1 -1883.222,E2 -1883.222} C_VEL
LIN {X 0,Y 580.139,Z 621.682,A -85,B 0,C 180,E1 -1884.439,E2 -1884.439} C_VEL
LIN {X 0,Y 580.108,Z 626.373,A -85,B 0,C 180,E1 -1885.484,E2 -1885.484} C_VEL
LIN {X 0,Y 580.123,Z 629.958,A -85,B 0,C 180,E1 -1886.528,E2 -1886.528} C_VEL
LIN {X 0,Y 580.043,Z 631.809,A -85,B 0,C 180,E1 -1887.222,E2 -1887.222} C_VEL
LIN {X 0,Y 580.038,Z 633.2,A -85,B 0,C 180,E1 -1887.917,E2 -1887.917} C_VEL
LIN {X 0,Y 580.04,Z 634.785,A -85,B 0,C 180,E1 -1889.306,E2 -1889.306} C_VEL
LIN {X 0,Y 580.037,Z 635,A -85,B 0,C 180,E1 -1890,E2 -1890} C_VEL
LIN {X 0,Y 580.047,Z 634.186,A -85,B 0,C 180,E1 -1891.389,E2 -1891.389} C_VEL
LIN {X 0,Y 580.038,Z 633.2,A -85,B 0,C 180,E1 -1892.083,E2 -1892.083} C_VEL
LIN {X 0,Y 580.043,Z 631.81,A -85,B 0,C 180,E1 -1892.778,E2 -1892.778} C_VEL
LIN {X 0,Y 580.109,Z 628.896,A -85,B 0,C 180,E1 -1893.821,E2 -1893.821} C_VEL
LIN {X 0,Y 580.054,Z 624.949,A -85,B 0,C 180,E1 -1894.865,E2 -1894.865} C_VEL
LIN {X 0,Y 580.139,Z 618.877,A -85,B 0,C 180,E1 -1896.085,E2 -1896.085} C_VEL
LIN {X 0,Y 580.184,Z 612.237,A -85,B 0,C 180,E1 -1897.132,E2 -1897.132} C_VEL
LIN {X 0,Y 580.25,Z 603.99,A -85,B 0,C 180,E1 -1898.182,E2 -1898.182} C_VEL
LIN {X 0,Y 580.308,Z 595.538,A -85,B 0,C 180,E1 -1899.058,E2 -1899.058} C_VEL
LIN {X 0,Y 580.417,Z 585.097,A -85,B 0,C 180,E1 -1899.936,E2 -1899.936} C_VEL
LIN {X 0,Y 580.495,Z 574.757,A -85,B 0,C 180,E1 -1900.64,E2 -1900.64} C_VEL
LIN {X 0,Y 580.597,Z 563.233,A -85,B 0,C 180,E1 -1901.265,E2 -1901.265} C_VEL
LIN {X 0,Y 580.674,Z 550.473,A -85,B 0,C 180,E1 -1901.785,E2 -1901.785} C_VEL
LIN {X 0,Y 580.775,Z 537.438,A -85,B 0,C 180,E1 -1902.159,E2 -1902.159} C_VEL
LIN {X 0,Y 580.849,Z 525.09,A -85,B 0,C 180,E1 -1902.38,E2 -1902.38} C_VEL
LIN {X 0,Y 580.908,Z 426.728,A -85,B 0,C 180,E1 -1903.601,E2 -1903.601} C_VEL
LIN {X 0,Y 580.388,Z 423.275,A -85,B 0,C 180,E1 -1903.68,E2 -1903.68} C_VEL
LIN {X 0,Y 580.51,Z 405.124,A -85,B 0,C 180,E1 -1906.348,E2 -1906.348} C_VEL
LIN {X 0,Y 580.646,Z 387.025,A -85,B 0,C 180,E1 -1909.075,E2 -1909.075} C_VEL
LIN {X 0,Y 580.829,Z 370.135,A -85,B 0,C 180,E1 -1911.656,E2 -1911.656} C_VEL
LIN {X 0,Y 580.313,Z 366.778,A -85,B 0,C 180,E1 -1912.238,E2 -1912.238} C_VEL
LIN {X 0,Y 580.311,Z 366.698,A -85,B 0,C 180,E1 -1915.079,E2 -1915.079} C_VEL
LIN {X 0,Y 580.3,Z 366.696,A -85,B 0,C 180,E1 -1918.185,E2 -1918.185} C_VEL
LIN {X 0,Y 580.294,Z 366.696,A -85,B 0,C 180,E1 -1920.696,E2 -1920.696} C_VEL
LIN {X 0,Y 580.305,Z 366.703,A -85,B 0,C 180,E1 -1923.316,E2 -1923.316} C_VEL
LIN {X 0,Y 580.327,Z 366.695,A -85,B 0,C 180,E1 -1925.767,E2 -1925.767} C_VEL
LIN {X 0,Y 580.289,Z 366.696,A -85,B 0,C 180,E1 -1928.146,E2 -1928.146} C_VEL
LIN {X 0,Y 580.3,Z 366.698,A -85,B 0,C 180,E1 -1930.843,E2 -1930.843} C_VEL
LIN {X 0,Y 580.286,Z 366.7,A -85,B 0,C 180,E1 -1933.656,E2 -1933.656} C_VEL
LIN {X 0,Y 580.29,Z 366.698,A -85,B 0,C 180,E1 -1936.607,E2 -1936.607} C_VEL
LIN {X 0,Y 580.318,Z 366.703,A -85,B 0,C 180,E1 -1939.158,E2 -1939.158} C_VEL
LIN {X 0,Y 580.289,Z 366.697,A -85,B 0,C 180,E1 -1941.926,E2 -1941.926} C_VEL
LIN {X 0,Y 580.303,Z 366.697,A -85,B 0,C 180,E1 -1944.456,E2 -1944.456} C_VEL
LIN {X 0,Y 580.289,Z 366.706,A -85,B 0,C 180,E1 -1946.975,E2 -1946.975} C_VEL
LIN {X 0,Y 580.298,Z 366.698,A -85,B 0,C 180,E1 -1949.425,E2 -1949.425} C_VEL
LIN {X 0,Y 580.315,Z 366.694,A -85,B 0,C 180,E1 -1952.136,E2 -1952.136} C_VEL
LIN {X 0,Y 580.302,Z 366.704,A -85,B 0,C 180,E1 -1954.92,E2 -1954.92} C_VEL
LIN {X 0,Y 580.27,Z 366.699,A -85,B 0,C 180,E1 -1957.947,E2 -1957.947} C_VEL
LIN {X 0,Y 580.312,Z 366.701,A -85,B 0,C 180,E1 -1960.914,E2 -1960.914} C_VEL
LIN {X 0,Y 580.277,Z 366.698,A -85,B 0,C 180,E1 -1963.825,E2 -1963.825} C_VEL
LIN {X 0,Y 580.319,Z 366.694,A -85,B 0,C 180,E1 -1965.983,E2 -1965.983} C_VEL
LIN {X 0,Y 580.297,Z 366.702,A -85,B 0,C 180,E1 -1968.827,E2 -1968.827} C_VEL
LIN {X 0,Y 580.328,Z 366.692,A -85,B 0,C 180,E1 -1971.644,E2 -1971.644} C_VEL
LIN {X 0,Y 580.318,Z 366.702,A -85,B 0,C 180,E1 -1974.44,E2 -1974.44} C_VEL
LIN {X 0,Y 580.34,Z 366.691,A -85,B 0,C 180,E1 -1977.223,E2 -1977.223} C_VEL
LIN {X 0,Y 580.345,Z 366.694,A -85,B 0,C 180,E1 -1980,E2 -1980} C_VEL
LIN {X 0,Y 580.34,Z 366.694,A -85,B 0,C 180,E1 -1982.776,E2 -1982.776} C_VEL
LIN {X 0,Y 580.32,Z 366.694,A -85,B 0,C 180,E1 -1985.56,E2 -1985.56} C_VEL
LIN {X 0,Y 580.329,Z 366.7,A -85,B 0,C 180,E1 -1988.356,E2 -1988.356} C_VEL
LIN {X 0,Y 580.292,Z 366.696,A -85,B 0,C 180,E1 -1991.191,E2 -1991.191} C_VEL
LIN {X 0,Y 580.32,Z 366.701,A -85,B 0,C 180,E1 -1994.017,E2 -1994.017} C_VEL
LIN {X 0,Y 580.309,Z 366.694,A -85,B 0,C 180,E1 -1996.916,E2 -1996.916} C_VEL
LIN {X 0,Y 580.303,Z 366.702,A -85,B 0,C 180,E1 -1999.822,E2 -1999.822} C_VEL
LIN {X 0,Y 580.283,Z 366.698,A -85,B 0,C 180,E1 -2001.342,E2 -2001.342} C_VEL
LIN {X 0,Y 579.586,Z 366.793,A -85,B 0,C 180,E1 -2001.921,E2 -2001.921} C_VEL
LIN {X 0,Y 576.709,Z 367.149,A -85,B 0,C 180,E1 -2002.861,E2 -2002.861} C_VEL
LIN {X 0,Y 574.313,Z 367.447,A -85,B 0,C 180,E1 -2003.617,E2 -2003.617} C_VEL
LIN {X 0,Y 573.314,Z 367.572,A -85,B 0,C 180,E1 -2004.201,E2 -2004.201} C_VEL
LIN {X 0,Y 573.247,Z 367.576,A -85,B 0,C 180,E1 -2004.398,E2 -2004.398} C_VEL
LIN {X 0,Y 573.259,Z 367.573,A -85,B 0,C 180,E1 -2006.976,E2 -2006.976} C_VEL
LIN {X 0,Y 573.25,Z 367.578,A -85,B 0,C 180,E1 -2009.49,E2 -2009.49} C_VEL
LIN {X 0,Y 573.253,Z 367.577,A -85,B 0,C 180,E1 -2012.23,E2 -2012.23} C_VEL
LIN {X 0,Y 573.247,Z 367.574,A -85,B 0,C 180,E1 -2014.774,E2 -2014.774} C_VEL
LIN {X 0,Y 573.251,Z 367.576,A -85,B 0,C 180,E1 -2017.167,E2 -2017.167} C_VEL
LIN {X 0,Y 573.245,Z 367.583,A -85,B 0,C 180,E1 -2019.607,E2 -2019.607} C_VEL
LIN {X 0,Y 573.241,Z 367.575,A -85,B 0,C 180,E1 -2022.643,E2 -2022.643} C_VEL
LIN {X 0,Y 573.232,Z 367.584,A -85,B 0,C 180,E1 -2025.667,E2 -2025.667} C_VEL
LIN {X 0,Y 573.243,Z 367.574,A -85,B 0,C 180,E1 -2028.545,E2 -2028.545} C_VEL
LIN {X 0,Y 573.248,Z 367.581,A -85,B 0,C 180,E1 -2031.3,E2 -2031.3} C_VEL
LIN {X 0,Y 573.264,Z 367.573,A -85,B 0,C 180,E1 -2034.012,E2 -2034.012} C_VEL
LIN {X 0,Y 573.285,Z 367.569,A -85,B 0,C 180,E1 -2036.519,E2 -2036.519} C_VEL
LIN {X 0,Y 573.234,Z 367.582,A -85,B 0,C 180,E1 -2039.117,E2 -2039.117} C_VEL
LIN {X 0,Y 573.252,Z 367.574,A -85,B 0,C 180,E1 -2041.971,E2 -2041.971} C_VEL
LIN {X 0,Y 573.255,Z 367.574,A -85,B 0,C 180,E1 -2044.59,E2 -2044.59} C_VEL
LIN {X 0,Y 573.236,Z 367.577,A -85,B 0,C 180,E1 -2047.662,E2 -2047.662} C_VEL
LIN {X 0,Y 573.267,Z 367.574,A -85,B 0,C 180,E1 -2050.67,E2 -2050.67} C_VEL
LIN {X 0,Y 573.249,Z 367.575,A -85,B 0,C 180,E1 -2053.622,E2 -2053.622} C_VEL
LIN {X 0,Y 573.276,Z 367.571,A -85,B 0,C 180,E1 -2055.807,E2 -2055.807} C_VEL
LIN {X 0,Y 573.265,Z 367.578,A -85,B 0,C 180,E1 -2058.745,E2 -2058.745} C_VEL
LIN {X 0,Y 573.286,Z 367.575,A -85,B 0,C 180,E1 -2061.541,E2 -2061.541} C_VEL
LIN {X 0,Y 573.305,Z 367.721,A -85,B 0,C 180,E1 -2062.339,E2 -2062.339} C_VEL
LIN {X 0,Y 573.686,Z 374.068,A -85,B 0,C 180,E1 -2063.442,E2 -2063.442} C_VEL
LIN {X 0,Y 573.494,Z 390.152,A -85,B 0,C 180,E1 -2066.135,E2 -2066.135} C_VEL
LIN {X 0,Y 573.343,Z 408.576,A -85,B 0,C 180,E1 -2069.166,E2 -2069.166} C_VEL
LIN {X 0,Y 573.494,Z 410,A -85,B 0,C 180,E1 -2069.243,E2 -2069.243} C_VEL
LIN {X 0,Y 574.073,Z 415.009,A -85,B 0,C 180,E1 -2069.32,E2 -2069.32} C_VEL
LIN {X 0,Y 573.873,Z 516.531,A -85,B 0,C 180,E1 -2070.614,E2 -2070.614} C_VEL
LIN {X 0,Y 573.809,Z 530.153,A -85,B 0,C 180,E1 -2070.943,E2 -2070.943} C_VEL
LIN {X 0,Y 573.651,Z 542.987,A -85,B 0,C 180,E1 -2071.404,E2 -2071.404} C_VEL
LIN {X 0,Y 573.538,Z 555.423,A -85,B 0,C 180,E1 -2072.019,E2 -2072.019} C_VEL
LIN {X 0,Y 573.422,Z 566.523,A -85,B 0,C 180,E1 -2072.722,E2 -2072.722} C_VEL
LIN {X 0,Y 573.325,Z 576.581,A -85,B 0,C 180,E1 -2073.514,E2 -2073.514} C_VEL
LIN {X 0,Y 573.224,Z 585.672,A -85,B 0,C 180,E1 -2074.395,E2 -2074.395} C_VEL
LIN {X 0,Y 573.091,Z 594.565,A -85,B 0,C 180,E1 -2075.453,E2 -2075.453} C_VEL
LIN {X 0,Y 573.066,Z 602.247,A -85,B 0,C 180,E1 -2076.6,E2 -2076.6} C_VEL
LIN {X 0,Y 573.022,Z 608.302,A -85,B 0,C 180,E1 -2077.753,E2 -2077.753} C_VEL
LIN {X 0,Y 573.001,Z 612.657,A -85,B 0,C 180,E1 -2078.819,E2 -2078.819} C_VEL
LIN {X 0,Y 572.98,Z 615.943,A -85,B 0,C 180,E1 -2079.887,E2 -2079.887} C_VEL
LIN {X 0,Y 572.983,Z 618.479,A -85,B 0,C 180,E1 -2081.112,E2 -2081.112} C_VEL
LIN {X 0,Y 572.946,Z 619.579,A -85,B 0,C 180,E1 -2082.036,E2 -2082.036} C_VEL
LIN {X 0,Y 572.945,Z 619.942,A -85,B 0,C 180,E1 -2082.755,E2 -2082.755} C_VEL
LIN {X 0,Y 572.968,Z 619.91,A -85,B 0,C 180,E1 -2083.476,E2 -2083.476} C_VEL
LIN {X 0,Y 572.961,Z 619.355,A -85,B 0,C 180,E1 -2084.298,E2 -2084.298} C_VEL
LIN {X 0,Y 572.933,Z 617.233,A -85,B 0,C 180,E1 -2085.656,E2 -2085.656} C_VEL
LIN {X 0,Y 572.993,Z 613.869,A -85,B 0,C 180,E1 -2086.922,E2 -2086.922} C_VEL
LIN {X 0,Y 572.999,Z 610.412,A -85,B 0,C 180,E1 -2087.856,E2 -2087.856} C_VEL
LIN {X 0,Y 573.065,Z 605.515,A -85,B 0,C 180,E1 -2088.903,E2 -2088.903} C_VEL
LIN {X 0,Y 573.09,Z 598.518,A -85,B 0,C 180,E1 -2090.082,E2 -2090.082} C_VEL
LIN {X 0,Y 573.157,Z 591.274,A -85,B 0,C 180,E1 -2091.056,E2 -2091.056} C_VEL
LIN {X 0,Y 573.251,Z 583.143,A -85,B 0,C 180,E1 -2091.957,E2 -2091.957} C_VEL
LIN {X 0,Y 573.384,Z 572.693,A -85,B 0,C 180,E1 -2092.902,E2 -2092.902} C_VEL
LIN {X 0,Y 573.475,Z 562.19,A -85,B 0,C 180,E1 -2093.663,E2 -2093.663} C_VEL
LIN {X 0,Y 573.58,Z 550.587,A -85,B 0,C 180,E1 -2094.33,E2 -2094.33} C_VEL
LIN {X 0,Y 573.74,Z 537.898,A -85,B 0,C 180,E1 -2094.888,E2 -2094.888} C_VEL
LIN {X 0,Y 573.84,Z 524.799,A -85,B 0,C 180,E1 -2095.296,E2 -2095.296} C_VEL
LIN {X 0,Y 573.9,Z 511.991,A -85,B 0,C 180,E1 -2095.549,E2 -2095.549} C_VEL
LIN {X 0,Y 574.047,Z 413.487,A -85,B 0,C 180,E1 -2096.79,E2 -2096.79} C_VEL
LIN {X 0,Y 573.339,Z 409.042,A -85,B 0,C 180,E1 -2096.883,E2 -2096.883} C_VEL
LIN {X 0,Y 573.351,Z 403.416,A -85,B 0,C 180,E1 -2097.761,E2 -2097.761} C_VEL
LIN {X 0,Y 573.495,Z 386.479,A -85,B 0,C 180,E1 -2100.568,E2 -2100.568} C_VEL
LIN {X 0,Y 573.665,Z 370.55,A -85,B 0,C 180,E1 -2103.245,E2 -2103.245} C_VEL
LIN {X 0,Y 573.271,Z 367.637,A -85,B 0,C 180,E1 -2103.801,E2 -2103.801} C_VEL
LIN {X 0,Y 573.259,Z 367.574,A -85,B 0,C 180,E1 -2106.047,E2 -2106.047} C_VEL
LIN {X 0,Y 573.248,Z 367.577,A -85,B 0,C 180,E1 -2108.7,E2 -2108.7} C_VEL
LIN {X 0,Y 573.25,Z 367.577,A -85,B 0,C 180,E1 -2111.595,E2 -2111.595} C_VEL
LIN {X 0,Y 573.234,Z 367.576,A -85,B 0,C 180,E1 -2114.332,E2 -2114.332} C_VEL
LIN {X 0,Y 573.256,Z 367.577,A -85,B 0,C 180,E1 -2117.355,E2 -2117.355} C_VEL
LIN {X 0,Y 573.245,Z 367.575,A -85,B 0,C 180,E1 -2120.393,E2 -2120.393} C_VEL
LIN {X 0,Y 573.251,Z 367.583,A -85,B 0,C 180,E1 -2123.077,E2 -2123.077} C_VEL
LIN {X 0,Y 573.268,Z 367.571,A -85,B 0,C 180,E1 -2125.671,E2 -2125.671} C_VEL
LIN {X 0,Y 573.244,Z 367.574,A -85,B 0,C 180,E1 -2128.185,E2 -2128.185} C_VEL
LIN {X 0,Y 573.263,Z 367.573,A -85,B 0,C 180,E1 -2130.634,E2 -2130.634} C_VEL
LIN {X 0,Y 573.265,Z 367.574,A -85,B 0,C 180,E1 -2133.499,E2 -2133.499} C_VEL
LIN {X 0,Y 573.236,Z 367.575,A -85,B 0,C 180,E1 -2136.135,E2 -2136.135} C_VEL
LIN {X 0,Y 573.251,Z 367.577,A -85,B 0,C 180,E1 -2138.706,E2 -2138.706} C_VEL
LIN {X 0,Y 573.232,Z 367.577,A -85,B 0,C 180,E1 -2141.412,E2 -2141.412} C_VEL
LIN {X 0,Y 573.253,Z 367.573,A -85,B 0,C 180,E1 -2143.622,E2 -2143.622} C_VEL
LIN {X 0,Y 573.233,Z 367.578,A -85,B 0,C 180,E1 -2146.529,E2 -2146.529} C_VEL
LIN {X 0,Y 573.268,Z 367.572,A -85,B 0,C 180,E1 -2149.403,E2 -2149.403} C_VEL
LIN {X 0,Y 573.282,Z 367.57,A -85,B 0,C 180,E1 -2152.25,E2 -2152.25} C_VEL
LIN {X 0,Y 573.307,Z 367.572,A -85,B 0,C 180,E1 -2155.077,E2 -2155.077} C_VEL
LIN {X 0,Y 573.301,Z 367.566,A -85,B 0,C 180,E1 -2157.892,E2 -2157.892} C_VEL
LIN {X 0,Y 573.334,Z 367.57,A -85,B 0,C 180,E1 -2160.702,E2 -2160.702} C_VEL
LIN {X 0,Y 573.237,Z 367.574,A -85,B 0,C 180,E1 -2163.515,E2 -2163.515} C_VEL
LIN {X 0,Y 573.287,Z 367.568,A -85,B 0,C 180,E1 -2165.628,E2 -2165.628} C_VEL
LIN {X 0,Y 573.3,Z 367.571,A -85,B 0,C 180,E1 -2168.459,E2 -2168.459} C_VEL
LIN {X 0,Y 573.289,Z 367.57,A -85,B 0,C 180,E1 -2171.312,E2 -2171.312} C_VEL
LIN {X 0,Y 573.272,Z 367.574,A -85,B 0,C 180,E1 -2174.425,E2 -2174.425} C_VEL
LIN {X 0,Y 573.253,Z 367.575,A -85,B 0,C 180,E1 -2177.112,E2 -2177.112} C_VEL
LIN {X 0,Y 573.251,Z 367.574,A -85,B 0,C 180,E1 -2180.077,E2 -2180.077} C_VEL
LIN {X 0,Y 573.263,Z 367.574,A -85,B 0,C 180,E1 -2183.154,E2 -2183.154} C_VEL
LIN {X 0,Y 573.282,Z 367.571,A -85,B 0,C 180,E1 -2186.189,E2 -2186.189} C_VEL
LIN {X 0,Y 573.237,Z 367.583,A -85,B 0,C 180,E1 -2188.565,E2 -2188.565} C_VEL
LIN {X 0,Y 573.231,Z 367.579,A -85,B 0,C 180,E1 -2190.993,E2 -2190.993} C_VEL
LIN {X 0,Y 573.281,Z 367.569,A -85,B 0,C 180,E1 -2193.529,E2 -2193.529} C_VEL
LIN {X 0,Y 573.255,Z 367.574,A -85,B 0,C 180,E1 -2196.049,E2 -2196.049} C_VEL
LIN {X 0,Y 573.244,Z 367.582,A -85,B 0,C 180,E1 -2198.702,E2 -2198.702} C_VEL
LIN {X 0,Y 573.261,Z 367.569,A -85,B 0,C 180,E1 -2201.598,E2 -2201.598} C_VEL
LIN {X 0,Y 573.235,Z 367.581,A -85,B 0,C 180,E1 -2204.334,E2 -2204.334} C_VEL
LIN {X 0,Y 573.239,Z 367.574,A -85,B 0,C 180,E1 -2207.359,E2 -2207.359} C_VEL
LIN {X 0,Y 573.246,Z 367.581,A -85,B 0,C 180,E1 -2210.394,E2 -2210.394} C_VEL
LIN {X 0,Y 573.255,Z 367.573,A -85,B 0,C 180,E1 -2213.079,E2 -2213.079} C_VEL
LIN {X 0,Y 573.274,Z 367.57,A -85,B 0,C 180,E1 -2215.673,E2 -2215.673} C_VEL
LIN {X 0,Y 573.249,Z 367.579,A -85,B 0,C 180,E1 -2218.186,E2 -2218.186} C_VEL
LIN {X 0,Y 573.266,Z 367.578,A -85,B 0,C 180,E1 -2220.635,E2 -2220.635} C_VEL
LIN {X 0,Y 573.27,Z 367.572,A -85,B 0,C 180,E1 -2223.501,E2 -2223.501} C_VEL
LIN {X 0,Y 573.233,Z 367.583,A -85,B 0,C 180,E1 -2226.135,E2 -2226.135} C_VEL
LIN {X 0,Y 573.308,Z 367.73,A -85,B 0,C 180,E1 -2227.642,E2 -2227.642} C_VEL
LIN {X 0,Y 573.86,Z 372.549,A -85,B 0,C 180,E1 -2228.445,E2 -2228.445} C_VEL
LIN {X 0,Y 573.675,Z 389.441,A -85,B 0,C 180,E1 -2231.056,E2 -2231.056} C_VEL
LIN {X 0,Y 573.493,Z 406.333,A -85,B 0,C 180,E1 -2233.629,E2 -2233.629} C_VEL
LIN {X 0,Y 573.376,Z 423.288,A -85,B 0,C 180,E1 -2236.149,E2 -2236.149} C_VEL
LIN {X 0,Y 574.094,Z 428.545,A -85,B 0,C 180,E1 -2236.257,E2 -2236.257} C_VEL
LIN {X 0,Y 573.893,Z 530.969,A -85,B 0,C 180,E1 -2237.558,E2 -2237.558} C_VEL
LIN {X 0,Y 573.833,Z 544.234,A -85,B 0,C 180,E1 -2237.871,E2 -2237.871} C_VEL
LIN {X 0,Y 573.717,Z 556.385,A -85,B 0,C 180,E1 -2238.295,E2 -2238.295} C_VEL
LIN {X 0,Y 573.576,Z 568.728,A -85,B 0,C 180,E1 -2238.879,E2 -2238.879} C_VEL
LIN {X 0,Y 573.431,Z 580.207,A -85,B 0,C 180,E1 -2239.585,E2 -2239.585} C_VEL
LIN {X 0,Y 573.328,Z 590.605,A -85,B 0,C 180,E1 -2240.386,E2 -2240.386} C_VEL
LIN {X 0,Y 573.241,Z 599.116,A -85,B 0,C 180,E1 -2241.185,E2 -2241.185} C_VEL
LIN {X 0,Y 573.161,Z 606.963,A -85,B 0,C 180,E1 -2242.071,E2 -2242.071} C_VEL
LIN {X 0,Y 573.072,Z 614.956,A -85,B 0,C 180,E1 -2243.186,E2 -2243.186} C_VEL
LIN {X 0,Y 573.07,Z 621.681,A -85,B 0,C 180,E1 -2244.37,E2 -2244.37} C_VEL
LIN {X 0,Y 573.029,Z 626.373,A -85,B 0,C 180,E1 -2245.428,E2 -2245.428} C_VEL
LIN {X 0,Y 573.022,Z 629.958,A -85,B 0,C 180,E1 -2246.484,E2 -2246.484} C_VEL
LIN {X 0,Y 572.959,Z 631.809,A -85,B 0,C 180,E1 -2247.188,E2 -2247.188} C_VEL
LIN {X 0,Y 572.938,Z 633.199,A -85,B 0,C 180,E1 -2247.891,E2 -2247.891} C_VEL
LIN {X 0,Y 572.94,Z 634.785,A -85,B 0,C 180,E1 -2249.297,E2 -2249.297} C_VEL
LIN {X 0,Y 572.938,Z 635,A -85,B 0,C 180,E1 -2250,E2 -2250} C_VEL
LIN {X 0,Y 572.946,Z 634.186,A -85,B 0,C 180,E1 -2251.406,E2 -2251.406} C_VEL
LIN {X 0,Y 572.938,Z 633.199,A -85,B 0,C 180,E1 -2252.109,E2 -2252.109} C_VEL
LIN {X 0,Y 572.959,Z 631.81,A -85,B 0,C 180,E1 -2252.812,E2 -2252.812} C_VEL
LIN {X 0,Y 573.014,Z 628.895,A -85,B 0,C 180,E1 -2253.868,E2 -2253.868} C_VEL
LIN {X 0,Y 572.963,Z 624.949,A -85,B 0,C 180,E1 -2254.926,E2 -2254.926} C_VEL
LIN {X 0,Y 573.064,Z 618.876,A -85,B 0,C 180,E1 -2256.16,E2 -2256.16} C_VEL
LIN {X 0,Y 573.119,Z 612.237,A -85,B 0,C 180,E1 -2257.221,E2 -2257.221} C_VEL
